LIN {X 0,Y 467.59,Z 413.241,A -85,B 0,C 180,E1 -7782.567,E2 -7782.567} C_VEL
LIN {X 0,Y 467.575,Z 413.244,A -85,B 0,C 180,E1 -7785.053,E2 -7785.053} C_VEL
LIN {X 0,Y 467.628,Z 413.238,A -85,B 0,C 180,E1 -7787.444,E2 -7787.444} C_VEL
LIN {X 0,Y 467.623,Z 413.239,A -85,B 0,C 180,E1 -7790.859,E2 -7790.859} C_VEL
LIN {X 0,Y 467.563,Z 413.244,A -85,B 0,C 180,E1 -7794.261,E2 -7794.261} C_VEL
LIN {X 0,Y 467.585,Z 413.242,A -85,B 0,C 180,E1 -7797.321,E2 -7797.321} C_VEL
LIN {X 0,Y 467.574,Z 413.245,A -85,B 0,C 180,E1 -7800.667,E2 -7800.667} C_VEL
LIN {X 0,Y 467.62,Z 413.238,A -85,B 0,C 180,E1 -7803.2,E2 -7803.2} C_VEL
LIN {X 0,Y 467.597,Z 413.241,A -85,B 0,C 180,E1 -7806.468,E2 -7806.468} C_VEL
LIN {X 0,Y 467.626,Z 413.235,A -85,B 0,C 180,E1 -7809.777,E2 -7809.777} C_VEL
LIN {X 0,Y 467.611,Z 413.24,A -85,B 0,C 180,E1 -7812.507,E2 -7812.507} C_VEL
LIN {X 0,Y 467.653,Z 413.233,A -85,B 0,C 180,E1 -7814.113,E2 -7814.113} C_VEL
LIN {X 0,Y 467.499,Z 414.001,A -85,B 0,C 180,E1 -7814.561,E2 -7814.561} C_VEL
LIN {X 0,Y 467.049,Z 415.884,A -85,B 0,C 180,E1 -7814.962,E2 -7814.962} C_VEL
LIN {X 0,Y 466.067,Z 420.004,A -85,B 0,C 180,E1 -7815.467,E2 -7815.467} C_VEL
LIN {X 0,Y 464.179,Z 429.024,A -85,B 0,C 180,E1 -7816.136,E2 -7816.136} C_VEL
LIN {X 0,Y 463.27,Z 436.592,A -85,B 0,C 180,E1 -7816.659,E2 -7816.659} C_VEL
LIN {X 0,Y 462.762,Z 447.595,A -85,B 0,C 180,E1 -7817.613,E2 -7817.613} C_VEL
LIN {X 0,Y 462.355,Z 456.798,A -85,B 0,C 180,E1 -7818.603,E2 -7818.603} C_VEL
LIN {X 0,Y 461.906,Z 465.182,A -85,B 0,C 180,E1 -7819.701,E2 -7819.701} C_VEL
LIN {X 0,Y 461.403,Z 473.311,A -85,B 0,C 180,E1 -7821.018,E2 -7821.018} C_VEL
LIN {X 0,Y 461.038,Z 479.446,A -85,B 0,C 180,E1 -7822.245,E2 -7822.245} C_VEL
LIN {X 0,Y 460.814,Z 485.803,A -85,B 0,C 180,E1 -7823.871,E2 -7823.871} C_VEL
LIN {X 0,Y 460.529,Z 489.69,A -85,B 0,C 180,E1 -7825.185,E2 -7825.185} C_VEL
LIN {X 0,Y 460.337,Z 492.556,A -85,B 0,C 180,E1 -7826.499,E2 -7826.499} C_VEL
LIN {X 0,Y 460.22,Z 493.935,A -85,B 0,C 180,E1 -7827.374,E2 -7827.374} C_VEL
LIN {X 0,Y 460.244,Z 494.899,A -85,B 0,C 180,E1 -7828.25,E2 -7828.25} C_VEL
LIN {X 0,Y 460.165,Z 495.736,A -85,B 0,C 180,E1 -7830,E2 -7830} C_VEL
LIN {X 0,Y 460.244,Z 494.978,A -85,B 0,C 180,E1 -7831.75,E2 -7831.75} C_VEL
LIN {X 0,Y 460.331,Z 492.716,A -85,B 0,C 180,E1 -7833.501,E2 -7833.501} C_VEL
LIN {X 0,Y 460.52,Z 489.91,A -85,B 0,C 180,E1 -7834.815,E2 -7834.815} C_VEL
LIN {X 0,Y 460.8,Z 486.099,A -85,B 0,C 180,E1 -7836.129,E2 -7836.129} C_VEL
LIN {X 0,Y 460.953,Z 480.215,A -85,B 0,C 180,E1 -7837.677,E2 -7837.677} C_VEL
LIN {X 0,Y 461.396,Z 473.809,A -85,B 0,C 180,E1 -7838.982,E2 -7838.982} C_VEL
LIN {X 0,Y 461.878,Z 465.789,A -85,B 0,C 180,E1 -7840.299,E2 -7840.299} C_VEL
LIN {X 0,Y 462.279,Z 457.573,A -85,B 0,C 180,E1 -7841.399,E2 -7841.399} C_VEL
LIN {X 0,Y 462.778,Z 447.396,A -85,B 0,C 180,E1 -7842.498,E2 -7842.498} C_VEL
LIN {X 0,Y 463.259,Z 436.893,A -85,B 0,C 180,E1 -7843.409,E2 -7843.409} C_VEL
LIN {X 0,Y 463.618,Z 426.234,A -85,B 0,C 180,E1 -7844.149,E2 -7844.149} C_VEL
LIN {X 0,Y 463.023,Z 422.562,A -85,B 0,C 180,E1 -7844.392,E2 -7844.392} C_VEL
LIN {X 0,Y 460.579,Z 414.111,A -85,B 0,C 180,E1 -7844.95,E2 -7844.95} C_VEL
LIN {X 0,Y 460.553,Z 414.12,A -85,B 0,C 180,E1 -7847.77,E2 -7847.77} C_VEL
LIN {X 0,Y 460.554,Z 414.117,A -85,B 0,C 180,E1 -7850.547,E2 -7850.547} C_VEL
LIN {X 0,Y 460.541,Z 414.12,A -85,B 0,C 180,E1 -7853.706,E2 -7853.706} C_VEL
LIN {X 0,Y 460.572,Z 414.114,A -85,B 0,C 180,E1 -7856.265,E2 -7856.265} C_VEL
LIN {X 0,Y 460.544,Z 414.12,A -85,B 0,C 180,E1 -7859.231,E2 -7859.231} C_VEL
LIN {X 0,Y 460.534,Z 414.118,A -85,B 0,C 180,E1 -7862.284,E2 -7862.284} C_VEL
LIN {X 0,Y 460.517,Z 414.123,A -85,B 0,C 180,E1 -7865.445,E2 -7865.445} C_VEL
LIN {X 0,Y 460.572,Z 414.116,A -85,B 0,C 180,E1 -7868.901,E2 -7868.901} C_VEL
LIN {X 0,Y 460.551,Z 414.116,A -85,B 0,C 180,E1 -7872.178,E2 -7872.178} C_VEL
LIN {X 0,Y 460.523,Z 414.122,A -85,B 0,C 180,E1 -7875.412,E2 -7875.412} C_VEL
LIN {X 0,Y 460.538,Z 414.119,A -85,B 0,C 180,E1 -7878.397,E2 -7878.397} C_VEL
LIN {X 0,Y 460.529,Z 414.121,A -85,B 0,C 180,E1 -7881.267,E2 -7881.267} C_VEL
LIN {X 0,Y 460.513,Z 414.123,A -85,B 0,C 180,E1 -7884.554,E2 -7884.554} C_VEL
LIN {X 0,Y 460.534,Z 414.118,A -85,B 0,C 180,E1 -7887.716,E2 -7887.716} C_VEL
LIN {X 0,Y 460.543,Z 414.12,A -85,B 0,C 180,E1 -7890.769,E2 -7890.769} C_VEL
LIN {X 0,Y 460.559,Z 414.115,A -85,B 0,C 180,E1 -7893.734,E2 -7893.734} C_VEL
LIN {X 0,Y 460.547,Z 414.12,A -85,B 0,C 180,E1 -7896.624,E2 -7896.624} C_VEL
LIN {X 0,Y 460.555,Z 414.116,A -85,B 0,C 180,E1 -7899.453,E2 -7899.453} C_VEL
LIN {X 0,Y 460.563,Z 414.118,A -85,B 0,C 180,E1 -7902.23,E2 -7902.23} C_VEL
LIN {X 0,Y 460.569,Z 414.117,A -85,B 0,C 180,E1 -7904.965,E2 -7904.965} C_VEL
LIN {X 0,Y 460.633,Z 414.106,A -85,B 0,C 180,E1 -7907.666,E2 -7907.666} C_VEL
LIN {X 0,Y 460.623,Z 414.108,A -85,B 0,C 180,E1 -7911.224,E2 -7911.224} C_VEL
LIN {X 0,Y 460.71,Z 414.098,A -85,B 0,C 180,E1 -7913.87,E2 -7913.87} C_VEL
LIN {X 0,Y 460.828,Z 414.081,A -85,B 0,C 180,E1 -7917.378,E2 -7917.378} C_VEL
LIN {X 0,Y 460.857,Z 414.08,A -85,B 0,C 180,E1 -7920,E2 -7920} C_VEL
LIN {X 0,Y 460.829,Z 414.084,A -85,B 0,C 180,E1 -7922.622,E2 -7922.622} C_VEL
LIN {X 0,Y 460.711,Z 414.099,A -85,B 0,C 180,E1 -7926.13,E2 -7926.13} C_VEL
LIN {X 0,Y 460.622,Z 414.109,A -85,B 0,C 180,E1 -7928.776,E2 -7928.776} C_VEL
LIN {X 0,Y 460.637,Z 414.109,A -85,B 0,C 180,E1 -7932.457,E2 -7932.457} C_VEL
LIN {X 0,Y 460.603,Z 414.114,A -85,B 0,C 180,E1 -7935.997,E2 -7935.997} C_VEL
LIN {X 0,Y 460.574,Z 414.114,A -85,B 0,C 180,E1 -7938.902,E2 -7938.902} C_VEL
LIN {X 0,Y 460.518,Z 414.122,A -85,B 0,C 180,E1 -7941.486,E2 -7941.486} C_VEL
LIN {X 0,Y 460.533,Z 414.121,A -85,B 0,C 180,E1 -7944.333,E2 -7944.333} C_VEL
LIN {X 0,Y 460.591,Z 414.115,A -85,B 0,C 180,E1 -7947.748,E2 -7947.748} C_VEL
LIN {X 0,Y 460.525,Z 414.12,A -85,B 0,C 180,E1 -7951.283,E2 -7951.283} C_VEL
LIN {X 0,Y 460.536,Z 414.12,A -85,B 0,C 180,E1 -7954.506,E2 -7954.506} C_VEL
LIN {X 0,Y 460.53,Z 414.121,A -85,B 0,C 180,E1 -7957.62,E2 -7957.62} C_VEL
LIN {X 0,Y 460.545,Z 414.119,A -85,B 0,C 180,E1 -7960.27,E2 -7960.27} C_VEL
LIN {X 0,Y 460.511,Z 414.125,A -85,B 0,C 180,E1 -7963.374,E2 -7963.374} C_VEL
LIN {X 0,Y 460.502,Z 414.127,A -85,B 0,C 180,E1 -7966.625,E2 -7966.625} C_VEL
LIN {X 0,Y 460.577,Z 414.173,A -85,B 0,C 180,E1 -7969.496,E2 -7969.496} C_VEL
LIN {X 0,Y 462.384,Z 423.509,A -85,B 0,C 180,E1 -7972.221,E2 -7972.221} C_VEL
LIN {X 0,Y 463.139,Z 428.94,A -85,B 0,C 180,E1 -7973.714,E2 -7973.714} C_VEL
LIN {X 0,Y 462.392,Z 443.333,A -85,B 0,C 180,E1 -7977.345,E2 -7977.345} C_VEL
LIN {X 0,Y 461.898,Z 456.337,A -85,B 0,C 180,E1 -7980.501,E2 -7980.501} C_VEL
LIN {X 0,Y 461.394,Z 471.111,A -85,B 0,C 180,E1 -7983.987,E2 -7983.987} C_VEL
LIN {X 0,Y 460.935,Z 485.612,A -85,B 0,C 180,E1 -7987.357,E2 -7987.357} C_VEL
LIN {X 0,Y 460.576,Z 500.515,A -85,B 0,C 180,E1 -7990.799,E2 -7990.799} C_VEL
LIN {X 0,Y 460.234,Z 515.613,A -85,B 0,C 180,E1 -7994.309,E2 -7994.309} C_VEL
LIN {X 0,Y 461.616,Z 530.277,A -85,B 0,C 180,E1 -7994.719,E2 -7994.719} C_VEL
LIN {X 0,Y 462.685,Z 543.371,A -85,B 0,C 180,E1 -7995.26,E2 -7995.26} C_VEL
LIN {X 0,Y 462.165,Z 555.697,A -85,B 0,C 180,E1 -7995.918,E2 -7995.918} C_VEL
LIN {X 0,Y 461.571,Z 568.295,A -85,B 0,C 180,E1 -7996.797,E2 -7996.797} C_VEL
LIN {X 0,Y 461.172,Z 579.391,A -85,B 0,C 180,E1 -7997.793,E2 -7997.793} C_VEL
LIN {X 0,Y 460.671,Z 588.435,A -85,B 0,C 180,E1 -7998.784,E2 -7998.784} C_VEL
LIN {X 0,Y 460.277,Z 598.303,A -85,B 0,C 180,E1 -8000.109,E2 -8000.109} C_VEL
LIN {X 0,Y 460.041,Z 606.193,A -85,B 0,C 180,E1 -8001.434,E2 -8001.434} C_VEL
LIN {X 0,Y 459.919,Z 613.486,A -85,B 0,C 180,E1 -8002.978,E2 -8002.978} C_VEL
LIN {X 0,Y 459.902,Z 618.355,A -85,B 0,C 180,E1 -8004.299,E2 -8004.299} C_VEL
LIN {X 0,Y 459.908,Z 622.081,A -85,B 0,C 180,E1 -8005.618,E2 -8005.618} C_VEL
LIN {X 0,Y 459.916,Z 624.005,A -85,B 0,C 180,E1 -8006.496,E2 -8006.496} C_VEL
LIN {X 0,Y 459.908,Z 625.446,A -85,B 0,C 180,E1 -8007.372,E2 -8007.372} C_VEL
LIN {X 0,Y 459.889,Z 626.473,A -85,B 0,C 180,E1 -8008.249,E2 -8008.249} C_VEL
LIN {X 0,Y 460.003,Z 627.34,A -85,B 0,C 180,E1 -8010,E2 -8010} C_VEL
LIN {X 0,Y 459.889,Z 626.474,A -85,B 0,C 180,E1 -8011.752,E2 -8011.752} C_VEL
LIN {X 0,Y 459.908,Z 625.45,A -85,B 0,C 180,E1 -8012.628,E2 -8012.628} C_VEL
LIN {X 0,Y 459.916,Z 624.008,A -85,B 0,C 180,E1 -8013.504,E2 -8013.504} C_VEL
LIN {X 0,Y 459.907,Z 620.977,A -85,B 0,C 180,E1 -8014.821,E2 -8014.821} C_VEL
LIN {X 0,Y 459.934,Z 616.882,A -85,B 0,C 180,E1 -8016.14,E2 -8016.14} C_VEL
LIN {X 0,Y 459.968,Z 610.586,A -85,B 0,C 180,E1 -8017.683,E2 -8017.683} C_VEL
LIN {X 0,Y 460.103,Z 603.731,A -85,B 0,C 180,E1 -8019.008,E2 -8019.008} C_VEL
LIN {X 0,Y 460.368,Z 595.255,A -85,B 0,C 180,E1 -8020.334,E2 -8020.334} C_VEL
LIN {X 0,Y 460.718,Z 586.591,A -85,B 0,C 180,E1 -8021.438,E2 -8021.438} C_VEL
LIN {X 0,Y 461.257,Z 576.549,A -85,B 0,C 180,E1 -8022.483,E2 -8022.483} C_VEL
LIN {X 0,Y 461.652,Z 566.849,A -85,B 0,C 180,E1 -8023.312,E2 -8023.312} C_VEL
LIN {X 0,Y 462.156,Z 555.684,A -85,B 0,C 180,E1 -8024.082,E2 -8024.082} C_VEL
LIN {X 0,Y 462.704,Z 543.348,A -85,B 0,C 180,E1 -8024.739,E2 -8024.739} C_VEL
LIN {X 0,Y 461.648,Z 530.24,A -85,B 0,C 180,E1 -8025.28,E2 -8025.28} C_VEL
LIN {X 0,Y 460.202,Z 515.503,A -85,B 0,C 180,E1 -8025.714,E2 -8025.714} C_VEL
LIN {X 0,Y 460.55,Z 501.845,A -85,B 0,C 180,E1 -8028.893,E2 -8028.893} C_VEL
LIN {X 0,Y 460.919,Z 486.637,A -85,B 0,C 180,E1 -8032.408,E2 -8032.408} C_VEL
LIN {X 0,Y 461.353,Z 472.748,A -85,B 0,C 180,E1 -8035.628,E2 -8035.628} C_VEL
LIN {X 0,Y 461.814,Z 457.82,A -85,B 0,C 180,E1 -8039.143,E2 -8039.143} C_VEL
LIN {X 0,Y 462.292,Z 445.378,A -85,B 0,C 180,E1 -8042.147,E2 -8042.147} C_VEL
LIN {X 0,Y 463.049,Z 430.956,A -85,B 0,C 180,E1 -8045.757,E2 -8045.757} C_VEL
LIN {X 0,Y 462.961,Z 426.694,A -85,B 0,C 180,E1 -8046.88,E2 -8046.88} C_VEL
LIN {X 0,Y 461.063,Z 416.459,A -85,B 0,C 180,E1 -8049.808,E2 -8049.808} C_VEL
LIN {X 0,Y 460.577,Z 414.114,A -85,B 0,C 180,E1 -8050.554,E2 -8050.554} C_VEL
LIN {X 0,Y 460.503,Z 414.123,A -85,B 0,C 180,E1 -8053.375,E2 -8053.375} C_VEL
LIN {X 0,Y 460.512,Z 414.126,A -85,B 0,C 180,E1 -8056.626,E2 -8056.626} C_VEL
LIN {X 0,Y 460.546,Z 414.119,A -85,B 0,C 180,E1 -8059.73,E2 -8059.73} C_VEL
LIN {X 0,Y 460.53,Z 414.121,A -85,B 0,C 180,E1 -8062.519,E2 -8062.519} C_VEL
LIN {X 0,Y 460.552,Z 414.118,A -85,B 0,C 180,E1 -8065.624,E2 -8065.624} C_VEL
LIN {X 0,Y 460.54,Z 414.118,A -85,B 0,C 180,E1 -8068.745,E2 -8068.745} C_VEL
LIN {X 0,Y 460.592,Z 414.115,A -85,B 0,C 180,E1 -8072.252,E2 -8072.252} C_VEL
LIN {X 0,Y 460.534,Z 414.121,A -85,B 0,C 180,E1 -8075.667,E2 -8075.667} C_VEL
LIN {X 0,Y 460.525,Z 414.121,A -85,B 0,C 180,E1 -8078.578,E2 -8078.578} C_VEL
LIN {X 0,Y 460.595,Z 414.113,A -85,B 0,C 180,E1 -8081.311,E2 -8081.311} C_VEL
LIN {X 0,Y 460.608,Z 414.113,A -85,B 0,C 180,E1 -8084.059,E2 -8084.059} C_VEL
LIN {X 0,Y 460.634,Z 414.109,A -85,B 0,C 180,E1 -8087.667,E2 -8087.667} C_VEL
LIN {X 0,Y 460.623,Z 414.109,A -85,B 0,C 180,E1 -8091.224,E2 -8091.224} C_VEL
LIN {X 0,Y 460.712,Z 414.099,A -85,B 0,C 180,E1 -8093.87,E2 -8093.87} C_VEL
LIN {X 0,Y 460.83,Z 414.084,A -85,B 0,C 180,E1 -8097.378,E2 -8097.378} C_VEL
LIN {X 0,Y 460.858,Z 414.08,A -85,B 0,C 180,E1 -8100,E2 -8100} C_VEL
LIN {X 0,Y 460.805,Z 414.084,A -85,B 0,C 180,E1 -8102.623,E2 -8102.623} C_VEL
LIN {X 0,Y 460.706,Z 414.099,A -85,B 0,C 180,E1 -8106.13,E2 -8106.13} C_VEL
LIN {X 0,Y 460.625,Z 414.108,A -85,B 0,C 180,E1 -8108.776,E2 -8108.776} C_VEL
LIN {X 0,Y 460.638,Z 414.105,A -85,B 0,C 180,E1 -8112.457,E2 -8112.457} C_VEL
LIN {X 0,Y 460.604,Z 414.111,A -85,B 0,C 180,E1 -8115.998,E2 -8115.998} C_VEL
LIN {X 0,Y 460.575,Z 414.115,A -85,B 0,C 180,E1 -8118.902,E2 -8118.902} C_VEL
LIN {X 0,Y 460.52,Z 414.123,A -85,B 0,C 180,E1 -8121.486,E2 -8121.486} C_VEL
LIN {X 0,Y 460.545,Z 414.117,A -85,B 0,C 180,E1 -8124.332,E2 -8124.332} C_VEL
LIN {X 0,Y 460.583,Z 414.115,A -85,B 0,C 180,E1 -8127.243,E2 -8127.243} C_VEL
LIN {X 0,Y 460.515,Z 414.12,A -85,B 0,C 180,E1 -8130.24,E2 -8130.24} C_VEL
LIN {X 0,Y 460.533,Z 414.121,A -85,B 0,C 180,E1 -8133.325,E2 -8133.325} C_VEL
LIN {X 0,Y 460.48,Z 414.127,A -85,B 0,C 180,E1 -8136.529,E2 -8136.529} C_VEL
LIN {X 0,Y 460.531,Z 414.119,A -85,B 0,C 180,E1 -8139.863,E2 -8139.863} C_VEL
LIN {X 0,Y 460.521,Z 414.123,A -85,B 0,C 180,E1 -8142.901,E2 -8142.901} C_VEL
LIN {X 0,Y 460.528,Z 414.119,A -85,B 0,C 180,E1 -8145.829,E2 -8145.829} C_VEL
LIN {X 0,Y 460.547,Z 414.12,A -85,B 0,C 180,E1 -8148.99,E2 -8148.99} C_VEL
LIN {X 0,Y 460.551,Z 414.119,A -85,B 0,C 180,E1 -8151.269,E2 -8151.269} C_VEL
LIN {X 0,Y 460.514,Z 414.124,A -85,B 0,C 180,E1 -8154.554,E2 -8154.554} C_VEL
LIN {X 0,Y 460.535,Z 414.118,A -85,B 0,C 180,E1 -8157.716,E2 -8157.716} C_VEL
LIN {X 0,Y 460.544,Z 414.121,A -85,B 0,C 180,E1 -8160.769,E2 -8160.769} C_VEL
LIN {X 0,Y 460.567,Z 414.115,A -85,B 0,C 180,E1 -8163.735,E2 -8163.735} C_VEL
LIN {X 0,Y 460.55,Z 414.119,A -85,B 0,C 180,E1 -8166.624,E2 -8166.624} C_VEL
LIN {X 0,Y 460.555,Z 414.117,A -85,B 0,C 180,E1 -8169.453,E2 -8169.453} C_VEL
LIN {X 0,Y 460.562,Z 414.119,A -85,B 0,C 180,E1 -8172.23,E2 -8172.23} C_VEL
LIN {X 0,Y 460.588,Z 414.114,A -85,B 0,C 180,E1 -8175.163,E2 -8175.163} C_VEL
LIN {X 0,Y 463.568,Z 424.775,A -85,B 0,C 180,E1 -8175.85,E2 -8175.85} C_VEL
LIN {X 0,Y 463.27,Z 436.592,A -85,B 0,C 180,E1 -8176.659,E2 -8176.659} C_VEL
LIN {X 0,Y 462.41,Z 441.639,A -85,B 0,C 180,E1 -8177.041,E2 -8177.041} C_VEL
LIN {X 0,Y 459.31,Z 449.618,A -85,B 0,C 180,E1 -8177.669,E2 -8177.669} C_VEL
LIN {X 0,Y 456.17,Z 457.098,A -85,B 0,C 180,E1 -8178.374,E2 -8178.374} C_VEL
LIN {X 0,Y 455.248,Z 461.313,A -85,B 0,C 180,E1 -8178.869,E2 -8178.869} C_VEL
LIN {X 0,Y 454.813,Z 469.099,A -85,B 0,C 180,E1 -8179.989,E2 -8179.989} C_VEL
LIN {X 0,Y 454.314,Z 476.678,A -85,B 0,C 180,E1 -8181.325,E2 -8181.325} C_VEL
LIN {X 0,Y 454.066,Z 481.966,A -85,B 0,C 180,E1 -8182.475,E2 -8182.475} C_VEL
LIN {X 0,Y 453.838,Z 486.808,A -85,B 0,C 180,E1 -8183.777,E2 -8183.777} C_VEL
LIN {X 0,Y 453.526,Z 490.696,A -85,B 0,C 180,E1 -8185.111,E2 -8185.111} C_VEL
LIN {X 0,Y 453.322,Z 493.562,A -85,B 0,C 180,E1 -8186.445,E2 -8186.445} C_VEL
LIN {X 0,Y 453.2,Z 494.941,A -85,B 0,C 180,E1 -8187.333,E2 -8187.333} C_VEL
LIN {X 0,Y 453.225,Z 495.903,A -85,B 0,C 180,E1 -8188.223,E2 -8188.223} C_VEL
LIN {X 0,Y 453.163,Z 496.737,A -85,B 0,C 180,E1 -8190,E2 -8190} C_VEL
LIN {X 0,Y 453.224,Z 495.982,A -85,B 0,C 180,E1 -8191.777,E2 -8191.777} C_VEL
LIN {X 0,Y 453.315,Z 493.721,A -85,B 0,C 180,E1 -8193.555,E2 -8193.555} C_VEL
LIN {X 0,Y 453.518,Z 490.914,A -85,B 0,C 180,E1 -8194.889,E2 -8194.889} C_VEL
LIN {X 0,Y 453.824,Z 487.101,A -85,B 0,C 180,E1 -8196.223,E2 -8196.223} C_VEL
LIN {X 0,Y 453.989,Z 481.22,A -85,B 0,C 180,E1 -8197.795,E2 -8197.795} C_VEL
LIN {X 0,Y 454.457,Z 474.811,A -85,B 0,C 180,E1 -8199.121,E2 -8199.121} C_VEL
LIN {X 0,Y 454.967,Z 466.791,A -85,B 0,C 180,E1 -8200.457,E2 -8200.457} C_VEL
LIN {X 0,Y 455.394,Z 458.574,A -85,B 0,C 180,E1 -8201.574,E2 -8201.574} C_VEL
LIN {X 0,Y 455.919,Z 448.396,A -85,B 0,C 180,E1 -8202.689,E2 -8202.689} C_VEL
LIN {X 0,Y 456.426,Z 437.892,A -85,B 0,C 180,E1 -8203.613,E2 -8203.613} C_VEL
LIN {X 0,Y 456.794,Z 427.234,A -85,B 0,C 180,E1 -8204.365,E2 -8204.365} C_VEL
LIN {X 0,Y 455.182,Z 420.664,A -85,B 0,C 180,E1 -8204.82,E2 -8204.82} C_VEL
LIN {X 0,Y 453.537,Z 414.991,A -85,B 0,C 180,E1 -8205.188,E2 -8205.188} C_VEL
LIN {X 0,Y 453.507,Z 414.997,A -85,B 0,C 180,E1 -8208.056,E2 -8208.056} C_VEL
LIN {X 0,Y 453.486,Z 414.998,A -85,B 0,C 180,E1 -8210.882,E2 -8210.882} C_VEL
LIN {X 0,Y 453.503,Z 414.996,A -85,B 0,C 180,E1 -8213.889,E2 -8213.889} C_VEL
LIN {X 0,Y 453.517,Z 414.994,A -85,B 0,C 180,E1 -8216.705,E2 -8216.705} C_VEL
LIN {X 0,Y 453.476,Z 414.998,A -85,B 0,C 180,E1 -8219.785,E2 -8219.785} C_VEL
LIN {X 0,Y 453.493,Z 414.998,A -85,B 0,C 180,E1 -8223.189,E2 -8223.189} C_VEL
LIN {X 0,Y 453.459,Z 415,A -85,B 0,C 180,E1 -8226.3,E2 -8226.3} C_VEL
LIN {X 0,Y 453.536,Z 414.992,A -85,B 0,C 180,E1 -8229.445,E2 -8229.445} C_VEL
LIN {X 0,Y 453.495,Z 414.998,A -85,B 0,C 180,E1 -8232.991,E2 -8232.991} C_VEL
LIN {X 0,Y 453.476,Z 414.997,A -85,B 0,C 180,E1 -8235.78,E2 -8235.78} C_VEL
LIN {X 0,Y 453.484,Z 414.997,A -85,B 0,C 180,E1 -8238.21,E2 -8238.21} C_VEL
LIN {X 0,Y 453.512,Z 414.997,A -85,B 0,C 180,E1 -8240.791,E2 -8240.791} C_VEL
LIN {X 0,Y 453.457,Z 415,A -85,B 0,C 180,E1 -8243.917,E2 -8243.917} C_VEL
LIN {X 0,Y 453.485,Z 414.999,A -85,B 0,C 180,E1 -8247.151,E2 -8247.151} C_VEL
LIN {X 0,Y 453.478,Z 414.998,A -85,B 0,C 180,E1 -8250.268,E2 -8250.268} C_VEL
LIN {X 0,Y 453.508,Z 414.995,A -85,B 0,C 180,E1 -8253.294,E2 -8253.294} C_VEL
LIN {X 0,Y 453.5,Z 414.996,A -85,B 0,C 180,E1 -8256.238,E2 -8256.238} C_VEL
LIN {X 0,Y 453.486,Z 414.998,A -85,B 0,C 180,E1 -8259.118,E2 -8259.118} C_VEL
LIN {X 0,Y 453.515,Z 414.993,A -85,B 0,C 180,E1 -8261.945,E2 -8261.945} C_VEL
LIN {X 0,Y 453.543,Z 414.992,A -85,B 0,C 180,E1 -8264.726,E2 -8264.726} C_VEL
LIN {X 0,Y 453.605,Z 414.981,A -85,B 0,C 180,E1 -8267.472,E2 -8267.472} C_VEL
LIN {X 0,Y 453.589,Z 414.985,A -85,B 0,C 180,E1 -8271.086,E2 -8271.086} C_VEL
LIN {X 0,Y 453.676,Z 414.973,A -85,B 0,C 180,E1 -8273.775,E2 -8273.775} C_VEL
LIN {X 0,Y 453.768,Z 414.961,A -85,B 0,C 180,E1 -8277.337,E2 -8277.337} C_VEL
LIN {X 0,Y 453.827,Z 414.956,A -85,B 0,C 180,E1 -8280,E2 -8280} C_VEL
LIN {X 0,Y 453.769,Z 414.964,A -85,B 0,C 180,E1 -8282.663,E2 -8282.663} C_VEL
LIN {X 0,Y 453.677,Z 414.976,A -85,B 0,C 180,E1 -8286.225,E2 -8286.225} C_VEL
LIN {X 0,Y 453.588,Z 414.985,A -85,B 0,C 180,E1 -8288.913,E2 -8288.913} C_VEL
LIN {X 0,Y 453.605,Z 414.984,A -85,B 0,C 180,E1 -8292.551,E2 -8292.551} C_VEL
LIN {X 0,Y 453.547,Z 414.992,A -85,B 0,C 180,E1 -8296.196,E2 -8296.196} C_VEL
LIN {X 0,Y 453.524,Z 414.992,A -85,B 0,C 180,E1 -8299.041,E2 -8299.041} C_VEL
LIN {X 0,Y 453.479,Z 415,A -85,B 0,C 180,E1 -8301.836,E2 -8301.836} C_VEL
LIN {X 0,Y 453.503,Z 414.995,A -85,B 0,C 180,E1 -8304.735,E2 -8304.735} C_VEL
LIN {X 0,Y 453.54,Z 414.993,A -85,B 0,C 180,E1 -8307.961,E2 -8307.961} C_VEL
LIN {X 0,Y 453.469,Z 415,A -85,B 0,C 180,E1 -8311.525,E2 -8311.525} C_VEL
LIN {X 0,Y 453.491,Z 414.996,A -85,B 0,C 180,E1 -8314.778,E2 -8314.778} C_VEL
LIN {X 0,Y 453.475,Z 414.999,A -85,B 0,C 180,E1 -8318.311,E2 -8318.311} C_VEL
LIN {X 0,Y 453.496,Z 414.995,A -85,B 0,C 180,E1 -8320.609,E2 -8320.609} C_VEL
LIN {X 0,Y 453.466,Z 415.003,A -85,B 0,C 180,E1 -8323.245,E2 -8323.245} C_VEL
LIN {X 0,Y 453.468,Z 415,A -85,B 0,C 180,E1 -8325.779,E2 -8325.779} C_VEL
LIN {X 0,Y 453.547,Z 415.09,A -85,B 0,C 180,E1 -8329.215,E2 -8329.215} C_VEL
LIN {X 0,Y 455.304,Z 424.201,A -85,B 0,C 180,E1 -8331.927,E2 -8331.927} C_VEL
LIN {X 0,Y 456.117,Z 428.865,A -85,B 0,C 180,E1 -8333.248,E2 -8333.248} C_VEL
LIN {X 0,Y 455.896,Z 434.726,A -85,B 0,C 180,E1 -8334.79,E2 -8334.79} C_VEL
LIN {X 0,Y 455.244,Z 448.739,A -85,B 0,C 180,E1 -8338.339,E2 -8338.339} C_VEL
LIN {X 0,Y 454.736,Z 461.139,A -85,B 0,C 180,E1 -8341.373,E2 -8341.373} C_VEL
LIN {X 0,Y 454.24,Z 474.519,A -85,B 0,C 180,E1 -8344.574,E2 -8344.574} C_VEL
LIN {X 0,Y 453.833,Z 487.75,A -85,B 0,C 180,E1 -8347.703,E2 -8347.703} C_VEL
LIN {X 0,Y 453.486,Z 501.768,A -85,B 0,C 180,E1 -8351.007,E2 -8351.007} C_VEL
LIN {X 0,Y 453.143,Z 514.766,A -85,B 0,C 180,E1 -8354.068,E2 -8354.068} C_VEL
LIN {X 0,Y 454.552,Z 528.842,A -85,B 0,C 180,E1 -8354.463,E2 -8354.463} C_VEL
LIN {X 0,Y 455.427,Z 539.753,A -85,B 0,C 180,E1 -8354.906,E2 -8354.906} C_VEL
LIN {X 0,Y 455.703,Z 544.635,A -85,B 0,C 180,E1 -8355.144,E2 -8355.144} C_VEL
LIN {X 0,Y 455.135,Z 556.46,A -85,B 0,C 180,E1 -8355.81,E2 -8355.81} C_VEL
LIN {X 0,Y 454.606,Z 567.274,A -85,B 0,C 180,E1 -8356.591,E2 -8356.591} C_VEL
LIN {X 0,Y 454.174,Z 578.369,A -85,B 0,C 180,E1 -8357.602,E2 -8357.602} C_VEL
LIN {X 0,Y 453.643,Z 587.412,A -85,B 0,C 180,E1 -8358.608,E2 -8358.608} C_VEL
LIN {X 0,Y 453.212,Z 597.279,A -85,B 0,C 180,E1 -8359.953,E2 -8359.953} C_VEL
LIN {X 0,Y 452.974,Z 605.172,A -85,B 0,C 180,E1 -8361.299,E2 -8361.299} C_VEL
LIN {X 0,Y 452.87,Z 610.593,A -85,B 0,C 180,E1 -8362.42,E2 -8362.42} C_VEL
LIN {X 0,Y 452.85,Z 615.865,A -85,B 0,C 180,E1 -8363.763,E2 -8363.763} C_VEL
LIN {X 0,Y 452.859,Z 619.965,A -85,B 0,C 180,E1 -8365.104,E2 -8365.104} C_VEL
LIN {X 0,Y 452.873,Z 622.996,A -85,B 0,C 180,E1 -8366.441,E2 -8366.441} C_VEL
LIN {X 0,Y 452.866,Z 624.438,A -85,B 0,C 180,E1 -8367.332,E2 -8367.332} C_VEL
LIN {X 0,Y 452.854,Z 625.466,A -85,B 0,C 180,E1 -8368.221,E2 -8368.221} C_VEL
LIN {X 0,Y 452.986,Z 626.337,A -85,B 0,C 180,E1 -8370,E2 -8370} C_VEL
LIN {X 0,Y 452.854,Z 625.468,A -85,B 0,C 180,E1 -8371.779,E2 -8371.779} C_VEL
LIN {X 0,Y 452.866,Z 624.441,A -85,B 0,C 180,E1 -8372.669,E2 -8372.669} C_VEL
LIN {X 0,Y 452.873,Z 622.999,A -85,B 0,C 180,E1 -8373.559,E2 -8373.559} C_VEL
LIN {X 0,Y 452.859,Z 619.966,A -85,B 0,C 180,E1 -8374.897,E2 -8374.897} C_VEL
LIN {X 0,Y 452.847,Z 615.862,A -85,B 0,C 180,E1 -8376.237,E2 -8376.237} C_VEL
LIN {X 0,Y 452.901,Z 609.565,A -85,B 0,C 180,E1 -8377.804,E2 -8377.804} C_VEL
LIN {X 0,Y 453.065,Z 602.711,A -85,B 0,C 180,E1 -8379.149,E2 -8379.149} C_VEL
LIN {X 0,Y 453.331,Z 594.231,A -85,B 0,C 180,E1 -8380.496,E2 -8380.496} C_VEL
LIN {X 0,Y 453.684,Z 585.563,A -85,B 0,C 180,E1 -8381.618,E2 -8381.618} C_VEL
LIN {X 0,Y 454.216,Z 576.067,A -85,B 0,C 180,E1 -8382.627,E2 -8382.627} C_VEL
LIN {X 0,Y 454.78,Z 564.38,A -85,B 0,C 180,E1 -8383.631,E2 -8383.631} C_VEL
LIN {X 0,Y 455.328,Z 552.874,A -85,B 0,C 180,E1 -8384.412,E2 -8384.412} C_VEL
LIN {X 0,Y 455.732,Z 542.312,A -85,B 0,C 180,E1 -8384.97,E2 -8384.97} C_VEL
LIN {X 0,Y 454.69,Z 530.257,A -85,B 0,C 180,E1 -8385.487,E2 -8385.487} C_VEL
LIN {X 0,Y 453.321,Z 516.581,A -85,B 0,C 180,E1 -8385.89,E2 -8385.89} C_VEL
LIN {X 0,Y 453.151,Z 514.574,A -85,B 0,C 180,E1 -8385.943,E2 -8385.943} C_VEL
LIN {X 0,Y 453.515,Z 499.972,A -85,B 0,C 180,E1 -8389.415,E2 -8389.415} C_VEL
LIN {X 0,Y 453.931,Z 484.708,A -85,B 0,C 180,E1 -8393.013,E2 -8393.013} C_VEL
LIN {X 0,Y 454.337,Z 471.213,A -85,B 0,C 180,E1 -8396.209,E2 -8396.209} C_VEL
LIN {X 0,Y 454.851,Z 458.02,A -85,B 0,C 180,E1 -8399.379,E2 -8399.379} C_VEL
LIN {X 0,Y 455.32,Z 446.381,A -85,B 0,C 180,E1 -8402.242,E2 -8402.242} C_VEL
LIN {X 0,Y 456.098,Z 432.25,A -85,B 0,C 180,E1 -8405.841,E2 -8405.841} C_VEL
LIN {X 0,Y 456.016,Z 428.134,A -85,B 0,C 180,E1 -8406.946,E2 -8406.946} C_VEL
LIN {X 0,Y 454.094,Z 417.758,A -85,B 0,C 180,E1 -8409.963,E2 -8409.963} C_VEL
LIN {X 0,Y 453.52,Z 414.995,A -85,B 0,C 180,E1 -8410.818,E2 -8410.818} C_VEL
LIN {X 0,Y 453.49,Z 415,A -85,B 0,C 180,E1 -8414.529,E2 -8414.529} C_VEL
LIN {X 0,Y 453.481,Z 415,A -85,B 0,C 180,E1 -8418.065,E2 -8418.065} C_VEL
LIN {X 0,Y 453.513,Z 414.994,A -85,B 0,C 180,E1 -8420.791,E2 -8420.791} C_VEL
LIN {X 0,Y 453.46,Z 415.003,A -85,B 0,C 180,E1 -8423.918,E2 -8423.918} C_VEL
LIN {X 0,Y 453.487,Z 414.996,A -85,B 0,C 180,E1 -8427.151,E2 -8427.151} C_VEL
LIN {X 0,Y 453.479,Z 415,A -85,B 0,C 180,E1 -8430.269,E2 -8430.269} C_VEL
LIN {X 0,Y 453.508,Z 414.994,A -85,B 0,C 180,E1 -8433.294,E2 -8433.294} C_VEL
LIN {X 0,Y 453.501,Z 414.997,A -85,B 0,C 180,E1 -8436.239,E2 -8436.239} C_VEL
LIN {X 0,Y 453.487,Z 414.997,A -85,B 0,C 180,E1 -8439.118,E2 -8439.118} C_VEL
LIN {X 0,Y 453.517,Z 414.997,A -85,B 0,C 180,E1 -8441.945,E2 -8441.945} C_VEL
LIN {X 0,Y 453.544,Z 414.988,A -85,B 0,C 180,E1 -8444.726,E2 -8444.726} C_VEL
LIN {X 0,Y 453.606,Z 414.984,A -85,B 0,C 180,E1 -8447.472,E2 -8447.472} C_VEL
LIN {X 0,Y 453.589,Z 414.984,A -85,B 0,C 180,E1 -8451.087,E2 -8451.087} C_VEL
LIN {X 0,Y 453.678,Z 414.976,A -85,B 0,C 180,E1 -8453.775,E2 -8453.775} C_VEL
LIN {X 0,Y 453.77,Z 414.964,A -85,B 0,C 180,E1 -8457.337,E2 -8457.337} C_VEL
LIN {X 0,Y 453.828,Z 414.956,A -85,B 0,C 180,E1 -8460,E2 -8460} C_VEL
LIN {X 0,Y 453.749,Z 414.963,A -85,B 0,C 180,E1 -8462.663,E2 -8462.663} C_VEL
LIN {X 0,Y 453.673,Z 414.974,A -85,B 0,C 180,E1 -8466.225,E2 -8466.225} C_VEL
LIN {X 0,Y 453.591,Z 414.985,A -85,B 0,C 180,E1 -8468.913,E2 -8468.913} C_VEL
LIN {X 0,Y 453.606,Z 414.981,A -85,B 0,C 180,E1 -8472.551,E2 -8472.551} C_VEL
LIN {X 0,Y 453.549,Z 414.988,A -85,B 0,C 180,E1 -8476.196,E2 -8476.196} C_VEL
LIN {X 0,Y 453.525,Z 414.994,A -85,B 0,C 180,E1 -8479.041,E2 -8479.041} C_VEL
LIN {X 0,Y 453.48,Z 414.999,A -85,B 0,C 180,E1 -8481.836,E2 -8481.836} C_VEL
LIN {X 0,Y 453.517,Z 414.994,A -85,B 0,C 180,E1 -8484.734,E2 -8484.734} C_VEL
LIN {X 0,Y 453.541,Z 414.99,A -85,B 0,C 180,E1 -8487.961,E2 -8487.961} C_VEL
LIN {X 0,Y 453.471,Z 415.001,A -85,B 0,C 180,E1 -8491.525,E2 -8491.525} C_VEL
LIN {X 0,Y 453.491,Z 414.997,A -85,B 0,C 180,E1 -8494.777,E2 -8494.777} C_VEL
LIN {X 0,Y 453.466,Z 414.999,A -85,B 0,C 180,E1 -8498.312,E2 -8498.312} C_VEL
LIN {X 0,Y 453.497,Z 414.997,A -85,B 0,C 180,E1 -8500.609,E2 -8500.609} C_VEL
LIN {X 0,Y 453.467,Z 415.002,A -85,B 0,C 180,E1 -8503.245,E2 -8503.245} C_VEL
LIN {X 0,Y 453.481,Z 414.997,A -85,B 0,C 180,E1 -8505.78,E2 -8505.78} C_VEL
LIN {X 0,Y 453.5,Z 414.995,A -85,B 0,C 180,E1 -8508.211,E2 -8508.211} C_VEL
LIN {X 0,Y 453.536,Z 414.993,A -85,B 0,C 180,E1 -8510.787,E2 -8510.787} C_VEL
LIN {X 0,Y 453.458,Z 415,A -85,B 0,C 180,E1 -8513.917,E2 -8513.917} C_VEL
LIN {X 0,Y 453.486,Z 415,A -85,B 0,C 180,E1 -8517.151,E2 -8517.151} C_VEL
LIN {X 0,Y 453.479,Z 414.998,A -85,B 0,C 180,E1 -8520.268,E2 -8520.268} C_VEL
LIN {X 0,Y 453.513,Z 414.995,A -85,B 0,C 180,E1 -8523.294,E2 -8523.294} C_VEL
LIN {X 0,Y 453.508,Z 414.995,A -85,B 0,C 180,E1 -8526.239,E2 -8526.239} C_VEL
LIN {X 0,Y 453.486,Z 414.998,A -85,B 0,C 180,E1 -8529.118,E2 -8529.118} C_VEL
LIN {X 0,Y 453.514,Z 414.996,A -85,B 0,C 180,E1 -8531.945,E2 -8531.945} C_VEL
LIN {X 0,Y 453.563,Z 415.113,A -85,B 0,C 180,E1 -8534.928,E2 -8534.928} C_VEL
LIN {X 0,Y 456.666,Z 425.801,A -85,B 0,C 180,E1 -8535.631,E2 -8535.631} C_VEL
LIN {X 0,Y 456.504,Z 436.314,A -85,B 0,C 180,E1 -8536.354,E2 -8536.354} C_VEL
LIN {X 0,Y 455.957,Z 447.451,A -85,B 0,C 180,E1 -8537.312,E2 -8537.312} C_VEL
LIN {X 0,Y 455.472,Z 457.806,A -85,B 0,C 180,E1 -8538.428,E2 -8538.428} C_VEL
LIN {X 0,Y 455.248,Z 461.313,A -85,B 0,C 180,E1 -8538.869,E2 -8538.869} C_VEL
LIN {X 0,Y 454.33,Z 465.42,A -85,B 0,C 180,E1 -8539.393,E2 -8539.393} C_VEL
LIN {X 0,Y 451.176,Z 471.828,A -85,B 0,C 180,E1 -8540.264,E2 -8540.264} C_VEL
LIN {X 0,Y 448.041,Z 477.616,A -85,B 0,C 180,E1 -8541.208,E2 -8541.208} C_VEL
LIN {X 0,Y 447.164,Z 480.748,A -85,B 0,C 180,E1 -8541.839,E2 -8541.839} C_VEL
LIN {X 0,Y 446.945,Z 486.257,A -85,B 0,C 180,E1 -8543.227,E2 -8543.227} C_VEL
LIN {X 0,Y 446.522,Z 490.514,A -85,B 0,C 180,E1 -8544.581,E2 -8544.581} C_VEL
LIN {X 0,Y 446.436,Z 492.744,A -85,B 0,C 180,E1 -8545.485,E2 -8545.485} C_VEL
LIN {X 0,Y 446.307,Z 494.568,A -85,B 0,C 180,E1 -8546.389,E2 -8546.389} C_VEL
LIN {X 0,Y 446.18,Z 495.946,A -85,B 0,C 180,E1 -8547.291,E2 -8547.291} C_VEL
LIN {X 0,Y 446.205,Z 496.908,A -85,B 0,C 180,E1 -8548.195,E2 -8548.195} C_VEL
LIN {X 0,Y 446.159,Z 497.739,A -85,B 0,C 180,E1 -8550,E2 -8550} C_VEL
LIN {X 0,Y 446.122,Z 497.563,A -85,B 0,C 180,E1 -8550.903,E2 -8550.903} C_VEL
LIN {X 0,Y 446.204,Z 496.986,A -85,B 0,C 180,E1 -8551.805,E2 -8551.805} C_VEL
LIN {X 0,Y 446.3,Z 494.725,A -85,B 0,C 180,E1 -8553.611,E2 -8553.611} C_VEL
LIN {X 0,Y 446.516,Z 491.919,A -85,B 0,C 180,E1 -8554.966,E2 -8554.966} C_VEL
LIN {X 0,Y 446.846,Z 488.103,A -85,B 0,C 180,E1 -8556.321,E2 -8556.321} C_VEL
LIN {X 0,Y 447.026,Z 482.225,A -85,B 0,C 180,E1 -8557.917,E2 -8557.917} C_VEL
LIN {X 0,Y 447.521,Z 475.813,A -85,B 0,C 180,E1 -8559.263,E2 -8559.263} C_VEL
LIN {X 0,Y 448.06,Z 467.793,A -85,B 0,C 180,E1 -8560.62,E2 -8560.62} C_VEL
LIN {X 0,Y 448.513,Z 459.576,A -85,B 0,C 180,E1 -8561.754,E2 -8561.754} C_VEL
LIN {X 0,Y 449.065,Z 449.397,A -85,B 0,C 180,E1 -8562.886,E2 -8562.886} C_VEL
LIN {X 0,Y 449.598,Z 438.891,A -85,B 0,C 180,E1 -8563.824,E2 -8563.824} C_VEL
LIN {X 0,Y 449.951,Z 428.238,A -85,B 0,C 180,E1 -8564.588,E2 -8564.588} C_VEL
LIN {X 0,Y 446.961,Z 417.622,A -85,B 0,C 180,E1 -8565.322,E2 -8565.322} C_VEL
LIN {X 0,Y 446.517,Z 415.865,A -85,B 0,C 180,E1 -8565.432,E2 -8565.432} C_VEL
LIN {X 0,Y 446.455,Z 415.874,A -85,B 0,C 180,E1 -8568.351,E2 -8568.351} C_VEL
LIN {X 0,Y 446.451,Z 415.875,A -85,B 0,C 180,E1 -8571.755,E2 -8571.755} C_VEL
LIN {X 0,Y 446.462,Z 415.874,A -85,B 0,C 180,E1 -8575.152,E2 -8575.152} C_VEL
LIN {X 0,Y 446.487,Z 415.868,A -85,B 0,C 180,E1 -8578.179,E2 -8578.179} C_VEL
LIN {X 0,Y 446.422,Z 415.877,A -85,B 0,C 180,E1 -8581.775,E2 -8581.775} C_VEL
LIN {X 0,Y 446.433,Z 415.875,A -85,B 0,C 180,E1 -8584.523,E2 -8584.523} C_VEL
LIN {X 0,Y 446.442,Z 415.874,A -85,B 0,C 180,E1 -8588.083,E2 -8588.083} C_VEL
LIN {X 0,Y 446.45,Z 415.876,A -85,B 0,C 180,E1 -8590.921,E2 -8590.921} C_VEL
LIN {X 0,Y 446.448,Z 415.872,A -85,B 0,C 180,E1 -8593.84,E2 -8593.84} C_VEL
LIN {X 0,Y 446.424,Z 415.876,A -85,B 0,C 180,E1 -8596.4,E2 -8596.4} C_VEL
LIN {X 0,Y 446.45,Z 415.873,A -85,B 0,C 180,E1 -8599.803,E2 -8599.803} C_VEL
LIN {X 0,Y 446.412,Z 415.878,A -85,B 0,C 180,E1 -8602.121,E2 -8602.121} C_VEL
LIN {X 0,Y 446.431,Z 415.876,A -85,B 0,C 180,E1 -8605.477,E2 -8605.477} C_VEL
LIN {X 0,Y 446.419,Z 415.88,A -85,B 0,C 180,E1 -8608.7,E2 -8608.7} C_VEL
LIN {X 0,Y 446.487,Z 415.867,A -85,B 0,C 180,E1 -8611.821,E2 -8611.821} C_VEL
LIN {X 0,Y 446.447,Z 415.876,A -85,B 0,C 180,E1 -8614.847,E2 -8614.847} C_VEL
LIN {X 0,Y 446.451,Z 415.875,A -85,B 0,C 180,E1 -8618.245,E2 -8618.245} C_VEL
LIN {X 0,Y 446.461,Z 415.871,A -85,B 0,C 180,E1 -8621.649,E2 -8621.649} C_VEL
LIN {X 0,Y 446.511,Z 415.868,A -85,B 0,C 180,E1 -8624.48,E2 -8624.48} C_VEL
LIN {X 0,Y 446.542,Z 415.863,A -85,B 0,C 180,E1 -8628.194,E2 -8628.194} C_VEL
LIN {X 0,Y 446.537,Z 415.864,A -85,B 0,C 180,E1 -8630.945,E2 -8630.945} C_VEL
LIN {X 0,Y 446.644,Z 415.849,A -85,B 0,C 180,E1 -8633.676,E2 -8633.676} C_VEL
LIN {X 0,Y 446.712,Z 415.84,A -85,B 0,C 180,E1 -8637.295,E2 -8637.295} C_VEL
LIN {X 0,Y 446.797,Z 415.831,A -85,B 0,C 180,E1 -8640,E2 -8640} C_VEL
LIN {X 0,Y 446.713,Z 415.843,A -85,B 0,C 180,E1 -8642.705,E2 -8642.705} C_VEL
LIN {X 0,Y 446.644,Z 415.853,A -85,B 0,C 180,E1 -8646.324,E2 -8646.324} C_VEL
LIN {X 0,Y 446.536,Z 415.862,A -85,B 0,C 180,E1 -8649.055,E2 -8649.055} C_VEL
LIN {X 0,Y 446.537,Z 415.863,A -85,B 0,C 180,E1 -8652.729,E2 -8652.729} C_VEL
LIN {X 0,Y 446.493,Z 415.87,A -85,B 0,C 180,E1 -8656.459,E2 -8656.459} C_VEL
LIN {X 0,Y 446.472,Z 415.87,A -85,B 0,C 180,E1 -8659.303,E2 -8659.303} C_VEL
LIN {X 0,Y 446.42,Z 415.88,A -85,B 0,C 180,E1 -8662.2,E2 -8662.2} C_VEL
LIN {X 0,Y 446.446,Z 415.873,A -85,B 0,C 180,E1 -8665.153,E2 -8665.153} C_VEL
LIN {X 0,Y 446.487,Z 415.871,A -85,B 0,C 180,E1 -8668.179,E2 -8668.179} C_VEL
LIN {X 0,Y 446.423,Z 415.879,A -85,B 0,C 180,E1 -8671.775,E2 -8671.775} C_VEL
LIN {X 0,Y 446.433,Z 415.876,A -85,B 0,C 180,E1 -8674.523,E2 -8674.523} C_VEL
LIN {X 0,Y 446.433,Z 415.878,A -85,B 0,C 180,E1 -8678.082,E2 -8678.082} C_VEL
LIN {X 0,Y 446.43,Z 415.875,A -85,B 0,C 180,E1 -8680.918,E2 -8680.918} C_VEL
LIN {X 0,Y 446.425,Z 415.879,A -85,B 0,C 180,E1 -8683.843,E2 -8683.843} C_VEL
LIN {X 0,Y 446.402,Z 415.882,A -85,B 0,C 180,E1 -8686.403,E2 -8686.403} C_VEL
LIN {X 0,Y 446.491,Z 415.952,A -85,B 0,C 180,E1 -8688.904,E2 -8688.904} C_VEL
LIN {X 0,Y 448.225,Z 424.909,A -85,B 0,C 180,E1 -8691.627,E2 -8691.627} C_VEL
LIN {X 0,Y 449.206,Z 430.494,A -85,B 0,C 180,E1 -8693.243,E2 -8693.243} C_VEL
LIN {X 0,Y 448.786,Z 438.672,A -85,B 0,C 180,E1 -8695.412,E2 -8695.412} C_VEL
LIN {X 0,Y 448.154,Z 452.05,A -85,B 0,C 180,E1 -8698.835,E2 -8698.835} C_VEL
LIN {X 0,Y 447.563,Z 465.435,A -85,B 0,C 180,E1 -8702.15,E2 -8702.15} C_VEL
LIN {X 0,Y 447.062,Z 478.722,A -85,B 0,C 180,E1 -8705.378,E2 -8705.378} C_VEL
LIN {X 0,Y 446.614,Z 492.854,A -85,B 0,C 180,E1 -8708.781,E2 -8708.781} C_VEL
LIN {X 0,Y 446.315,Z 504.726,A -85,B 0,C 180,E1 -8711.643,E2 -8711.643} C_VEL
LIN {X 0,Y 446.094,Z 513.582,A -85,B 0,C 180,E1 -8713.795,E2 -8713.795} C_VEL
LIN {X 0,Y 447.609,Z 528.964,A -85,B 0,C 180,E1 -8714.252,E2 -8714.252} C_VEL
LIN {X 0,Y 448.569,Z 541.291,A -85,B 0,C 180,E1 -8714.786,E2 -8714.786} C_VEL
LIN {X 0,Y 448.639,Z 547.933,A -85,B 0,C 180,E1 -8715.137,E2 -8715.137} C_VEL
LIN {X 0,Y 447.948,Z 560.356,A -85,B 0,C 180,E1 -8715.925,E2 -8715.925} C_VEL
LIN {X 0,Y 447.408,Z 570.845,A -85,B 0,C 180,E1 -8716.774,E2 -8716.774} C_VEL
LIN {X 0,Y 447.011,Z 580.591,A -85,B 0,C 180,E1 -8717.746,E2 -8717.746} C_VEL
LIN {X 0,Y 446.445,Z 589.924,A -85,B 0,C 180,E1 -8718.881,E2 -8718.881} C_VEL
LIN {X 0,Y 446.055,Z 599.061,A -85,B 0,C 180,E1 -8720.249,E2 -8720.249} C_VEL
LIN {X 0,Y 445.858,Z 606.448,A -85,B 0,C 180,E1 -8721.616,E2 -8721.616} C_VEL
LIN {X 0,Y 445.776,Z 611.449,A -85,B 0,C 180,E1 -8722.754,E2 -8722.754} C_VEL
LIN {X 0,Y 445.786,Z 616.327,A -85,B 0,C 180,E1 -8724.118,E2 -8724.118} C_VEL
LIN {X 0,Y 445.812,Z 620.06,A -85,B 0,C 180,E1 -8725.479,E2 -8725.479} C_VEL
LIN {X 0,Y 445.831,Z 621.987,A -85,B 0,C 180,E1 -8726.385,E2 -8726.385} C_VEL
LIN {X 0,Y 445.823,Z 623.43,A -85,B 0,C 180,E1 -8727.289,E2 -8727.289} C_VEL
LIN {X 0,Y 445.819,Z 624.459,A -85,B 0,C 180,E1 -8728.193,E2 -8728.193} C_VEL
LIN {X 0,Y 445.968,Z 625.333,A -85,B 0,C 180,E1 -8730,E2 -8730} C_VEL
LIN {X 0,Y 445.819,Z 624.461,A -85,B 0,C 180,E1 -8731.807,E2 -8731.807} C_VEL
LIN {X 0,Y 445.823,Z 623.433,A -85,B 0,C 180,E1 -8732.711,E2 -8732.711} C_VEL
LIN {X 0,Y 445.831,Z 621.989,A -85,B 0,C 180,E1 -8733.615,E2 -8733.615} C_VEL
LIN {X 0,Y 445.81,Z 618.953,A -85,B 0,C 180,E1 -8734.974,E2 -8734.974} C_VEL
LIN {X 0,Y 445.758,Z 613.74,A -85,B 0,C 180,E1 -8736.643,E2 -8736.643} C_VEL
LIN {X 0,Y 445.861,Z 607.505,A -85,B 0,C 180,E1 -8738.156,E2 -8738.156} C_VEL
LIN {X 0,Y 446.036,Z 600.418,A -85,B 0,C 180,E1 -8739.523,E2 -8739.523} C_VEL
LIN {X 0,Y 446.369,Z 591.581,A -85,B 0,C 180,E1 -8740.891,E2 -8740.891} C_VEL
LIN {X 0,Y 446.832,Z 582.56,A -85,B 0,C 180,E1 -8742.029,E2 -8742.029} C_VEL
LIN {X 0,Y 447.307,Z 571.973,A -85,B 0,C 180,E1 -8743.121,E2 -8743.121} C_VEL
LIN {X 0,Y 447.862,Z 561.901,A -85,B 0,C 180,E1 -8743.962,E2 -8743.962} C_VEL
LIN {X 0,Y 448.513,Z 549.9,A -85,B 0,C 180,E1 -8744.752,E2 -8744.752} C_VEL
LIN {X 0,Y 448.703,Z 542.412,A -85,B 0,C 180,E1 -8745.152,E2 -8745.152} C_VEL
LIN {X 0,Y 447.767,Z 530.864,A -85,B 0,C 180,E1 -8745.673,E2 -8745.673} C_VEL
LIN {X 0,Y 446.535,Z 517.889,A -85,B 0,C 180,E1 -8746.092,E2 -8746.092} C_VEL
LIN {X 0,Y 446.082,Z 513.649,A -85,B 0,C 180,E1 -8746.19,E2 -8746.19} C_VEL
LIN {X 0,Y 446.402,Z 500.788,A -85,B 0,C 180,E1 -8749.306,E2 -8749.306} C_VEL
LIN {X 0,Y 446.843,Z 485.819,A -85,B 0,C 180,E1 -8752.909,E2 -8752.909} C_VEL
LIN {X 0,Y 447.285,Z 472.599,A -85,B 0,C 180,E1 -8756.101,E2 -8756.101} C_VEL
LIN {X 0,Y 447.811,Z 459.234,A -85,B 0,C 180,E1 -8759.37,E2 -8759.37} C_VEL
LIN {X 0,Y 448.38,Z 446.873,A -85,B 0,C 180,E1 -8762.469,E2 -8762.469} C_VEL
LIN {X 0,Y 449.169,Z 433.473,A -85,B 0,C 180,E1 -8765.943,E2 -8765.943} C_VEL
LIN {X 0,Y 449.072,Z 429.445,A -85,B 0,C 180,E1 -8767.046,E2 -8767.046} C_VEL
LIN {X 0,Y 447.131,Z 419.044,A -85,B 0,C 180,E1 -8770.124,E2 -8770.124} C_VEL
LIN {X 0,Y 446.472,Z 415.874,A -85,B 0,C 180,E1 -8771.119,E2 -8771.119} C_VEL
LIN {X 0,Y 446.457,Z 415.874,A -85,B 0,C 180,E1 -8774.897,E2 -8774.897} C_VEL
LIN {X 0,Y 446.439,Z 415.877,A -85,B 0,C 180,E1 -8777.722,E2 -8777.722} C_VEL
LIN {X 0,Y 446.46,Z 415.871,A -85,B 0,C 180,E1 -8780.974,E2 -8780.974} C_VEL
LIN {X 0,Y 446.424,Z 415.878,A -85,B 0,C 180,E1 -8784.374,E2 -8784.374} C_VEL
LIN {X 0,Y 446.426,Z 415.879,A -85,B 0,C 180,E1 -8787.639,E2 -8787.639} C_VEL
LIN {X 0,Y 446.453,Z 415.872,A -85,B 0,C 180,E1 -8790.791,E2 -8790.791} C_VEL
LIN {X 0,Y 446.481,Z 415.872,A -85,B 0,C 180,E1 -8793.849,E2 -8793.849} C_VEL
LIN {X 0,Y 446.43,Z 415.875,A -85,B 0,C 180,E1 -8796.823,E2 -8796.823} C_VEL
LIN {X 0,Y 446.449,Z 415.876,A -85,B 0,C 180,E1 -8799.737,E2 -8799.737} C_VEL
LIN {X 0,Y 446.468,Z 415.871,A -85,B 0,C 180,E1 -8802.597,E2 -8802.597} C_VEL
LIN {X 0,Y 446.474,Z 415.872,A -85,B 0,C 180,E1 -8805.413,E2 -8805.413} C_VEL
LIN {X 0,Y 446.543,Z 415.863,A -85,B 0,C 180,E1 -8808.194,E2 -8808.194} C_VEL
LIN {X 0,Y 446.537,Z 415.862,A -85,B 0,C 180,E1 -8810.945,E2 -8810.945} C_VEL
LIN {X 0,Y 446.645,Z 415.852,A -85,B 0,C 180,E1 -8813.676,E2 -8813.676} C_VEL
LIN {X 0,Y 446.714,Z 415.843,A -85,B 0,C 180,E1 -8817.295,E2 -8817.295} C_VEL
LIN {X 0,Y 446.798,Z 415.831,A -85,B 0,C 180,E1 -8820,E2 -8820} C_VEL
LIN {X 0,Y 446.696,Z 415.841,A -85,B 0,C 180,E1 -8822.705,E2 -8822.705} C_VEL
LIN {X 0,Y 446.641,Z 415.849,A -85,B 0,C 180,E1 -8826.324,E2 -8826.324} C_VEL
LIN {X 0,Y 446.538,Z 415.864,A -85,B 0,C 180,E1 -8829.055,E2 -8829.055} C_VEL
LIN {X 0,Y 446.538,Z 415.862,A -85,B 0,C 180,E1 -8832.729,E2 -8832.729} C_VEL
LIN {X 0,Y 446.494,Z 415.866,A -85,B 0,C 180,E1 -8836.459,E2 -8836.459} C_VEL
LIN {X 0,Y 446.474,Z 415.874,A -85,B 0,C 180,E1 -8839.303,E2 -8839.303} C_VEL
LIN {X 0,Y 446.422,Z 415.876,A -85,B 0,C 180,E1 -8842.2,E2 -8842.2} C_VEL
LIN {X 0,Y 446.461,Z 415.874,A -85,B 0,C 180,E1 -8845.152,E2 -8845.152} C_VEL
LIN {X 0,Y 446.488,Z 415.867,A -85,B 0,C 180,E1 -8848.179,E2 -8848.179} C_VEL
LIN {X 0,Y 446.424,Z 415.877,A -85,B 0,C 180,E1 -8851.775,E2 -8851.775} C_VEL
LIN {X 0,Y 446.432,Z 415.876,A -85,B 0,C 180,E1 -8854.523,E2 -8854.523} C_VEL
LIN {X 0,Y 446.418,Z 415.877,A -85,B 0,C 180,E1 -8858.079,E2 -8858.079} C_VEL
LIN {X 0,Y 446.431,Z 415.878,A -85,B 0,C 180,E1 -8860.918,E2 -8860.918} C_VEL
LIN {X 0,Y 446.426,Z 415.875,A -85,B 0,C 180,E1 -8863.843,E2 -8863.843} C_VEL
LIN {X 0,Y 446.451,Z 415.873,A -85,B 0,C 180,E1 -8866.397,E2 -8866.397} C_VEL
LIN {X 0,Y 446.473,Z 415.87,A -85,B 0,C 180,E1 -8869.805,E2 -8869.805} C_VEL
LIN {X 0,Y 446.437,Z 415.874,A -85,B 0,C 180,E1 -8872.124,E2 -8872.124} C_VEL
LIN {X 0,Y 446.432,Z 415.876,A -85,B 0,C 180,E1 -8875.477,E2 -8875.477} C_VEL
LIN {X 0,Y 446.42,Z 415.88,A -85,B 0,C 180,E1 -8878.7,E2 -8878.7} C_VEL
LIN {X 0,Y 446.488,Z 415.867,A -85,B 0,C 180,E1 -8881.821,E2 -8881.821} C_VEL
LIN {X 0,Y 446.462,Z 415.875,A -85,B 0,C 180,E1 -8884.848,E2 -8884.848} C_VEL
LIN {X 0,Y 446.452,Z 415.874,A -85,B 0,C 180,E1 -8888.245,E2 -8888.245} C_VEL
LIN {X 0,Y 446.46,Z 415.873,A -85,B 0,C 180,E1 -8891.649,E2 -8891.649} C_VEL
LIN {X 0,Y 446.504,Z 415.869,A -85,B 0,C 180,E1 -8894.655,E2 -8894.655} C_VEL
LIN {X 0,Y 449.7,Z 426.838,A -85,B 0,C 180,E1 -8895.404,E2 -8895.404} C_VEL
LIN {X 0,Y 449.944,Z 429.876,A -85,B 0,C 180,E1 -8895.614,E2 -8895.614} C_VEL
LIN {X 0,Y 449.446,Z 440.976,A -85,B 0,C 180,E1 -8896.434,E2 -8896.434} C_VEL
LIN {X 0,Y 448.915,Z 451.829,A -85,B 0,C 180,E1 -8897.454,E2 -8897.454} C_VEL
LIN {X 0,Y 448.356,Z 462.355,A -85,B 0,C 180,E1 -8898.7,E2 -8898.7} C_VEL
LIN {X 0,Y 447.896,Z 470.107,A -85,B 0,C 180,E1 -8899.832,E2 -8899.832} C_VEL
LIN {X 0,Y 447.368,Z 477.685,A -85,B 0,C 180,E1 -8901.189,E2 -8901.189} C_VEL
LIN {X 0,Y 447.164,Z 480.748,A -85,B 0,C 180,E1 -8901.839,E2 -8901.839} C_VEL
LIN {X 0,Y 446.299,Z 483.671,A -85,B 0,C 180,E1 -8902.49,E2 -8902.49} C_VEL
LIN {X 0,Y 443.227,Z 488.126,A -85,B 0,C 180,E1 -8903.562,E2 -8903.562} C_VEL
LIN {X 0,Y 440.205,Z 491.913,A -85,B 0,C 180,E1 -8904.686,E2 -8904.686} C_VEL
LIN {X 0,Y 439.43,Z 493.743,A -85,B 0,C 180,E1 -8905.41,E2 -8905.41} C_VEL
LIN {X 0,Y 439.293,Z 495.574,A -85,B 0,C 180,E1 -8906.331,E2 -8906.331} C_VEL
LIN {X 0,Y 439.16,Z 496.952,A -85,B 0,C 180,E1 -8907.248,E2 -8907.248} C_VEL
LIN {X 0,Y 439.184,Z 497.913,A -85,B 0,C 180,E1 -8908.166,E2 -8908.166} C_VEL
LIN {X 0,Y 439.152,Z 498.741,A -85,B 0,C 180,E1 -8910,E2 -8910} C_VEL
LIN {X 0,Y 439.099,Z 498.567,A -85,B 0,C 180,E1 -8910.917,E2 -8910.917} C_VEL
LIN {X 0,Y 439.184,Z 497.99,A -85,B 0,C 180,E1 -8911.834,E2 -8911.834} C_VEL
LIN {X 0,Y 439.286,Z 495.73,A -85,B 0,C 180,E1 -8913.669,E2 -8913.669} C_VEL
LIN {X 0,Y 439.516,Z 492.922,A -85,B 0,C 180,E1 -8915.045,E2 -8915.045} C_VEL
LIN {X 0,Y 439.868,Z 489.106,A -85,B 0,C 180,E1 -8916.421,E2 -8916.421} C_VEL
LIN {X 0,Y 440.066,Z 483.229,A -85,B 0,C 180,E1 -8918.042,E2 -8918.042} C_VEL
LIN {X 0,Y 440.588,Z 476.816,A -85,B 0,C 180,E1 -8919.41,E2 -8919.41} C_VEL
LIN {X 0,Y 441.157,Z 468.795,A -85,B 0,C 180,E1 -8920.789,E2 -8920.789} C_VEL
LIN {X 0,Y 441.635,Z 460.577,A -85,B 0,C 180,E1 -8921.939,E2 -8921.939} C_VEL
LIN {X 0,Y 442.216,Z 450.398,A -85,B 0,C 180,E1 -8923.089,E2 -8923.089} C_VEL
LIN {X 0,Y 442.777,Z 439.891,A -85,B 0,C 180,E1 -8924.042,E2 -8924.042} C_VEL
LIN {X 0,Y 443.064,Z 429.249,A -85,B 0,C 180,E1 -8924.82,E2 -8924.82} C_VEL
LIN {X 0,Y 439.564,Z 417.335,A -85,B 0,C 180,E1 -8925.653,E2 -8925.653} C_VEL
LIN {X 0,Y 439.471,Z 416.743,A -85,B 0,C 180,E1 -8925.716,E2 -8925.716} C_VEL
LIN {X 0,Y 439.444,Z 416.749,A -85,B 0,C 180,E1 -8929.337,E2 -8929.337} C_VEL
LIN {X 0,Y 439.369,Z 416.755,A -85,B 0,C 180,E1 -8932.575,E2 -8932.575} C_VEL
LIN {X 0,Y 439.409,Z 416.752,A -85,B 0,C 180,E1 -8935.585,E2 -8935.585} C_VEL
LIN {X 0,Y 439.42,Z 416.749,A -85,B 0,C 180,E1 -8938.673,E2 -8938.673} C_VEL
LIN {X 0,Y 439.373,Z 416.753,A -85,B 0,C 180,E1 -8942.03,E2 -8942.03} C_VEL
LIN {X 0,Y 439.399,Z 416.754,A -85,B 0,C 180,E1 -8945.341,E2 -8945.341} C_VEL
LIN {X 0,Y 439.402,Z 416.752,A -85,B 0,C 180,E1 -8948.593,E2 -8948.593} C_VEL
LIN {X 0,Y 439.408,Z 416.753,A -85,B 0,C 180,E1 -8951.259,E2 -8951.259} C_VEL
LIN {X 0,Y 439.412,Z 416.753,A -85,B 0,C 180,E1 -8954.728,E2 -8954.728} C_VEL
LIN {X 0,Y 439.4,Z 416.75,A -85,B 0,C 180,E1 -8957.796,E2 -8957.796} C_VEL
LIN {X 0,Y 439.432,Z 416.747,A -85,B 0,C 180,E1 -8960.228,E2 -8960.228} C_VEL
LIN {X 0,Y 439.376,Z 416.754,A -85,B 0,C 180,E1 -8963.713,E2 -8963.713} C_VEL
LIN {X 0,Y 439.375,Z 416.757,A -85,B 0,C 180,E1 -8967.054,E2 -8967.054} C_VEL
LIN {X 0,Y 439.385,Z 416.753,A -85,B 0,C 180,E1 -8970.274,E2 -8970.274} C_VEL
LIN {X 0,Y 439.432,Z 416.747,A -85,B 0,C 180,E1 -8973.396,E2 -8973.396} C_VEL
LIN {X 0,Y 439.387,Z 416.755,A -85,B 0,C 180,E1 -8976.429,E2 -8976.429} C_VEL
LIN {X 0,Y 439.392,Z 416.752,A -85,B 0,C 180,E1 -8979.397,E2 -8979.397} C_VEL
LIN {X 0,Y 439.435,Z 416.749,A -85,B 0,C 180,E1 -8982.31,E2 -8982.31} C_VEL
LIN {X 0,Y 439.451,Z 416.745,A -85,B 0,C 180,E1 -8985.174,E2 -8985.174} C_VEL
LIN {X 0,Y 439.511,Z 416.738,A -85,B 0,C 180,E1 -8988.002,E2 -8988.002} C_VEL
LIN {X 0,Y 439.507,Z 416.738,A -85,B 0,C 180,E1 -8991.725,E2 -8991.725} C_VEL
LIN {X 0,Y 439.623,Z 416.727,A -85,B 0,C 180,E1 -8994.496,E2 -8994.496} C_VEL
LIN {X 0,Y 439.639,Z 416.725,A -85,B 0,C 180,E1 -8998.168,E2 -8998.168} C_VEL
LIN {X 0,Y 439.767,Z 416.707,A -85,B 0,C 180,E1 -9000,E2 -9000} C_VEL
LIN {X 0,Y 439.66,Z 416.721,A -85,B 0,C 180,E1 -9002.749,E2 -9002.749} C_VEL
LIN {X 0,Y 439.616,Z 416.727,A -85,B 0,C 180,E1 -9006.425,E2 -9006.425} C_VEL
LIN {X 0,Y 439.499,Z 416.738,A -85,B 0,C 180,E1 -9009.202,E2 -9009.202} C_VEL
LIN {X 0,Y 439.507,Z 416.738,A -85,B 0,C 180,E1 -9012.726,E2 -9012.726} C_VEL
LIN {X 0,Y 439.45,Z 416.748,A -85,B 0,C 180,E1 -9016.349,E2 -9016.349} C_VEL
LIN {X 0,Y 439.405,Z 416.752,A -85,B 0,C 180,E1 -9019.626,E2 -9019.626} C_VEL
LIN {X 0,Y 439.366,Z 416.757,A -85,B 0,C 180,E1 -9022.575,E2 -9022.575} C_VEL
LIN {X 0,Y 439.4,Z 416.752,A -85,B 0,C 180,E1 -9025.585,E2 -9025.585} C_VEL
LIN {X 0,Y 439.42,Z 416.748,A -85,B 0,C 180,E1 -9028.673,E2 -9028.673} C_VEL
LIN {X 0,Y 439.373,Z 416.757,A -85,B 0,C 180,E1 -9032.031,E2 -9032.031} C_VEL
LIN {X 0,Y 439.398,Z 416.752,A -85,B 0,C 180,E1 -9035.341,E2 -9035.341} C_VEL
LIN {X 0,Y 439.391,Z 416.752,A -85,B 0,C 180,E1 -9038.594,E2 -9038.594} C_VEL
LIN {X 0,Y 439.391,Z 416.752,A -85,B 0,C 180,E1 -9041.257,E2 -9041.257} C_VEL
LIN {X 0,Y 439.407,Z 416.756,A -85,B 0,C 180,E1 -9044.729,E2 -9044.729} C_VEL
LIN {X 0,Y 439.438,Z 416.849,A -85,B 0,C 180,E1 -9048.596,E2 -9048.596} C_VEL
LIN {X 0,Y 441.349,Z 426.573,A -85,B 0,C 180,E1 -9051.608,E2 -9051.608} C_VEL
LIN {X 0,Y 442.312,Z 432.803,A -85,B 0,C 180,E1 -9053.427,E2 -9053.427} C_VEL
LIN {X 0,Y 441.513,Z 446.095,A -85,B 0,C 180,E1 -9056.962,E2 -9056.962} C_VEL
LIN {X 0,Y 440.876,Z 458.439,A -85,B 0,C 180,E1 -9060.128,E2 -9060.128} C_VEL
LIN {X 0,Y 440.343,Z 471.318,A -85,B 0,C 180,E1 -9063.352,E2 -9063.352} C_VEL
LIN {X 0,Y 439.795,Z 485.911,A -85,B 0,C 180,E1 -9066.951,E2 -9066.951} C_VEL
LIN {X 0,Y 439.366,Z 499.836,A -85,B 0,C 180,E1 -9070.372,E2 -9070.372} C_VEL
LIN {X 0,Y 439.021,Z 512.588,A -85,B 0,C 180,E1 -9073.533,E2 -9073.533} C_VEL
LIN {X 0,Y 440.53,Z 527.398,A -85,B 0,C 180,E1 -9073.975,E2 -9073.975} C_VEL
LIN {X 0,Y 441.467,Z 540.244,A -85,B 0,C 180,E1 -9074.535,E2 -9074.535} C_VEL
LIN {X 0,Y 441.751,Z 546.918,A -85,B 0,C 180,E1 -9074.899,E2 -9074.899} C_VEL
LIN {X 0,Y 440.991,Z 559.333,A -85,B 0,C 180,E1 -9075.699,E2 -9075.699} C_VEL
LIN {X 0,Y 440.408,Z 570.09,A -85,B 0,C 180,E1 -9076.585,E2 -9076.585} C_VEL
LIN {X 0,Y 440.027,Z 579.57,A -85,B 0,C 180,E1 -9077.548,E2 -9077.548} C_VEL
LIN {X 0,Y 439.426,Z 588.903,A -85,B 0,C 180,E1 -9078.701,E2 -9078.701} C_VEL
LIN {X 0,Y 438.995,Z 598.038,A -85,B 0,C 180,E1 -9080.09,E2 -9080.09} C_VEL
LIN {X 0,Y 438.795,Z 605.428,A -85,B 0,C 180,E1 -9081.48,E2 -9081.48} C_VEL
LIN {X 0,Y 438.707,Z 610.431,A -85,B 0,C 180,E1 -9082.637,E2 -9082.637} C_VEL
LIN {X 0,Y 438.725,Z 615.312,A -85,B 0,C 180,E1 -9084.023,E2 -9084.023} C_VEL
LIN {X 0,Y 438.767,Z 619.049,A -85,B 0,C 180,E1 -9085.406,E2 -9085.406} C_VEL
LIN {X 0,Y 438.79,Z 620.978,A -85,B 0,C 180,E1 -9086.327,E2 -9086.327} C_VEL
LIN {X 0,Y 438.781,Z 622.422,A -85,B 0,C 180,E1 -9087.246,E2 -9087.246} C_VEL
LIN {X 0,Y 438.783,Z 623.453,A -85,B 0,C 180,E1 -9088.164,E2 -9088.164} C_VEL
LIN {X 0,Y 438.948,Z 624.329,A -85,B 0,C 180,E1 -9090,E2 -9090} C_VEL
LIN {X 0,Y 438.783,Z 623.454,A -85,B 0,C 180,E1 -9091.836,E2 -9091.836} C_VEL
LIN {X 0,Y 438.781,Z 622.424,A -85,B 0,C 180,E1 -9092.754,E2 -9092.754} C_VEL
LIN {X 0,Y 438.79,Z 620.98,A -85,B 0,C 180,E1 -9093.673,E2 -9093.673} C_VEL
LIN {X 0,Y 438.761,Z 617.941,A -85,B 0,C 180,E1 -9095.054,E2 -9095.054} C_VEL
LIN {X 0,Y 438.686,Z 613.095,A -85,B 0,C 180,E1 -9096.647,E2 -9096.647} C_VEL
LIN {X 0,Y 438.777,Z 606.481,A -85,B 0,C 180,E1 -9098.288,E2 -9098.288} C_VEL
LIN {X 0,Y 438.969,Z 599.392,A -85,B 0,C 180,E1 -9099.678,E2 -9099.678} C_VEL
LIN {X 0,Y 439.334,Z 590.554,A -85,B 0,C 180,E1 -9101.068,E2 -9101.068} C_VEL
LIN {X 0,Y 439.863,Z 581.538,A -85,B 0,C 180,E1 -9102.222,E2 -9102.222} C_VEL
LIN {X 0,Y 440.284,Z 571.825,A -85,B 0,C 180,E1 -9103.248,E2 -9103.248} C_VEL
LIN {X 0,Y 440.921,Z 560.874,A -85,B 0,C 180,E1 -9104.186,E2 -9104.186} C_VEL
LIN {X 0,Y 441.629,Z 548.877,A -85,B 0,C 180,E1 -9104.987,E2 -9104.987} C_VEL
LIN {X 0,Y 441.681,Z 542.513,A -85,B 0,C 180,E1 -9105.34,E2 -9105.34} C_VEL
LIN {X 0,Y 440.733,Z 530.049,A -85,B 0,C 180,E1 -9105.92,E2 -9105.92} C_VEL
LIN {X 0,Y 439.472,Z 516.795,A -85,B 0,C 180,E1 -9106.359,E2 -9106.359} C_VEL
LIN {X 0,Y 439.028,Z 512.565,A -85,B 0,C 180,E1 -9106.467,E2 -9106.467} C_VEL
LIN {X 0,Y 439.361,Z 499.818,A -85,B 0,C 180,E1 -9109.628,E2 -9109.628} C_VEL
LIN {X 0,Y 439.809,Z 484.892,A -85,B 0,C 180,E1 -9113.297,E2 -9113.297} C_VEL
LIN {X 0,Y 440.316,Z 471.332,A -85,B 0,C 180,E1 -9116.641,E2 -9116.641} C_VEL
LIN {X 0,Y 440.876,Z 458.416,A -85,B 0,C 180,E1 -9119.871,E2 -9119.871} C_VEL
LIN {X 0,Y 441.509,Z 446.064,A -85,B 0,C 180,E1 -9123.038,E2 -9123.038} C_VEL
LIN {X 0,Y 442.306,Z 432.765,A -85,B 0,C 180,E1 -9126.574,E2 -9126.574} C_VEL
LIN {X 0,Y 441.142,Z 425.574,A -85,B 0,C 180,E1 -9128.681,E2 -9128.681} C_VEL
LIN {X 0,Y 439.422,Z 416.749,A -85,B 0,C 180,E1 -9131.438,E2 -9131.438} C_VEL
LIN {X 0,Y 439.408,Z 416.751,A -85,B 0,C 180,E1 -9135.271,E2 -9135.271} C_VEL
LIN {X 0,Y 439.393,Z 416.757,A -85,B 0,C 180,E1 -9138.743,E2 -9138.743} C_VEL
LIN {X 0,Y 439.388,Z 416.754,A -85,B 0,C 180,E1 -9141.606,E2 -9141.606} C_VEL
LIN {X 0,Y 439.404,Z 416.75,A -85,B 0,C 180,E1 -9144.844,E2 -9144.844} C_VEL
LIN {X 0,Y 439.377,Z 416.758,A -85,B 0,C 180,E1 -9148.14,E2 -9148.14} C_VEL
LIN {X 0,Y 439.436,Z 416.748,A -85,B 0,C 180,E1 -9151.598,E2 -9151.598} C_VEL
LIN {X 0,Y 439.401,Z 416.752,A -85,B 0,C 180,E1 -9154.415,E2 -9154.415} C_VEL
LIN {X 0,Y 439.367,Z 416.756,A -85,B 0,C 180,E1 -9157.425,E2 -9157.425} C_VEL
LIN {X 0,Y 439.445,Z 416.745,A -85,B 0,C 180,E1 -9160.663,E2 -9160.663} C_VEL
LIN {X 0,Y 439.466,Z 416.744,A -85,B 0,C 180,E1 -9164.225,E2 -9164.225} C_VEL
LIN {X 0,Y 439.511,Z 416.74,A -85,B 0,C 180,E1 -9168.002,E2 -9168.002} C_VEL
LIN {X 0,Y 439.507,Z 416.741,A -85,B 0,C 180,E1 -9171.726,E2 -9171.726} C_VEL
LIN {X 0,Y 439.624,Z 416.723,A -85,B 0,C 180,E1 -9174.496,E2 -9174.496} C_VEL
LIN {X 0,Y 439.641,Z 416.722,A -85,B 0,C 180,E1 -9178.168,E2 -9178.168} C_VEL
LIN {X 0,Y 439.768,Z 416.707,A -85,B 0,C 180,E1 -9180,E2 -9180} C_VEL
LIN {X 0,Y 439.645,Z 416.72,A -85,B 0,C 180,E1 -9182.749,E2 -9182.749} C_VEL
LIN {X 0,Y 439.614,Z 416.724,A -85,B 0,C 180,E1 -9186.425,E2 -9186.425} C_VEL
LIN {X 0,Y 439.501,Z 416.741,A -85,B 0,C 180,E1 -9189.202,E2 -9189.202} C_VEL
LIN {X 0,Y 439.508,Z 416.737,A -85,B 0,C 180,E1 -9192.727,E2 -9192.727} C_VEL
LIN {X 0,Y 439.451,Z 416.743,A -85,B 0,C 180,E1 -9196.349,E2 -9196.349} C_VEL
LIN {X 0,Y 439.407,Z 416.753,A -85,B 0,C 180,E1 -9199.626,E2 -9199.626} C_VEL
LIN {X 0,Y 439.369,Z 416.755,A -85,B 0,C 180,E1 -9202.575,E2 -9202.575} C_VEL
LIN {X 0,Y 439.409,Z 416.752,A -85,B 0,C 180,E1 -9205.585,E2 -9205.585} C_VEL
LIN {X 0,Y 439.421,Z 416.749,A -85,B 0,C 180,E1 -9208.673,E2 -9208.673} C_VEL
LIN {X 0,Y 439.374,Z 416.754,A -85,B 0,C 180,E1 -9212.031,E2 -9212.031} C_VEL
LIN {X 0,Y 439.398,Z 416.754,A -85,B 0,C 180,E1 -9215.34,E2 -9215.34} C_VEL
LIN {X 0,Y 439.38,Z 416.755,A -85,B 0,C 180,E1 -9218.595,E2 -9218.595} C_VEL
LIN {X 0,Y 439.393,Z 416.756,A -85,B 0,C 180,E1 -9221.257,E2 -9221.257} C_VEL
LIN {X 0,Y 439.41,Z 416.752,A -85,B 0,C 180,E1 -9224.728,E2 -9224.728} C_VEL
LIN {X 0,Y 439.416,Z 416.749,A -85,B 0,C 180,E1 -9227.798,E2 -9227.798} C_VEL
LIN {X 0,Y 439.456,Z 416.744,A -85,B 0,C 180,E1 -9230.23,E2 -9230.23} C_VEL
LIN {X 0,Y 439.379,Z 416.753,A -85,B 0,C 180,E1 -9233.713,E2 -9233.713} C_VEL
LIN {X 0,Y 439.376,Z 416.758,A -85,B 0,C 180,E1 -9237.054,E2 -9237.054} C_VEL
LIN {X 0,Y 439.386,Z 416.753,A -85,B 0,C 180,E1 -9240.274,E2 -9240.274} C_VEL
LIN {X 0,Y 439.433,Z 416.748,A -85,B 0,C 180,E1 -9243.396,E2 -9243.396} C_VEL
LIN {X 0,Y 439.391,Z 416.754,A -85,B 0,C 180,E1 -9246.43,E2 -9246.43} C_VEL
LIN {X 0,Y 439.392,Z 416.752,A -85,B 0,C 180,E1 -9249.397,E2 -9249.397} C_VEL
LIN {X 0,Y 439.434,Z 416.75,A -85,B 0,C 180,E1 -9252.309,E2 -9252.309} C_VEL
LIN {X 0,Y 439.491,Z 416.9,A -85,B 0,C 180,E1 -9254.419,E2 -9254.419} C_VEL
LIN {X 0,Y 442.738,Z 427.875,A -85,B 0,C 180,E1 -9255.169,E2 -9255.169} C_VEL
LIN {X 0,Y 443.148,Z 430.99,A -85,B 0,C 180,E1 -9255.396,E2 -9255.396} C_VEL
LIN {X 0,Y 442.621,Z 441.986,A -85,B 0,C 180,E1 -9256.221,E2 -9256.221} C_VEL
LIN {X 0,Y 442.058,Z 452.839,A -85,B 0,C 180,E1 -9257.256,E2 -9257.256} C_VEL
LIN {X 0,Y 441.47,Z 463.363,A -85,B 0,C 180,E1 -9258.522,E2 -9258.522} C_VEL
LIN {X 0,Y 440.983,Z 471.114,A -85,B 0,C 180,E1 -9259.671,E2 -9259.671} C_VEL
LIN {X 0,Y 440.425,Z 478.692,A -85,B 0,C 180,E1 -9261.049,E2 -9261.049} C_VEL
LIN {X 0,Y 440.137,Z 483.972,A -85,B 0,C 180,E1 -9262.233,E2 -9262.233} C_VEL
LIN {X 0,Y 439.885,Z 488.819,A -85,B 0,C 180,E1 -9263.579,E2 -9263.579} C_VEL
LIN {X 0,Y 439.523,Z 492.708,A -85,B 0,C 180,E1 -9264.954,E2 -9264.954} C_VEL
LIN {X 0,Y 439.43,Z 493.743,A -85,B 0,C 180,E1 -9265.41,E2 -9265.41} C_VEL
LIN {X 0,Y 438.651,Z 495.37,A -85,B 0,C 180,E1 -9266.145,E2 -9266.145} C_VEL
LIN {X 0,Y 435.652,Z 497.663,A -85,B 0,C 180,E1 -9267.349,E2 -9267.349} C_VEL
LIN {X 0,Y 432.73,Z 499.192,A -85,B 0,C 180,E1 -9268.585,E2 -9268.585} C_VEL
LIN {X 0,Y 432.084,Z 499.594,A -85,B 0,C 180,E1 -9269.362,E2 -9269.362} C_VEL
LIN {X 0,Y 432.075,Z 499.572,A -85,B 0,C 180,E1 -9270.932,E2 -9270.932} C_VEL
LIN {X 0,Y 432.163,Z 498.994,A -85,B 0,C 180,E1 -9271.864,E2 -9271.864} C_VEL
LIN {X 0,Y 432.272,Z 496.734,A -85,B 0,C 180,E1 -9273.729,E2 -9273.729} C_VEL
LIN {X 0,Y 432.517,Z 493.926,A -85,B 0,C 180,E1 -9275.127,E2 -9275.127} C_VEL
LIN {X 0,Y 432.889,Z 490.109,A -85,B 0,C 180,E1 -9276.525,E2 -9276.525} C_VEL
LIN {X 0,Y 433.108,Z 484.234,A -85,B 0,C 180,E1 -9278.172,E2 -9278.172} C_VEL
LIN {X 0,Y 433.659,Z 477.818,A -85,B 0,C 180,E1 -9279.562,E2 -9279.562} C_VEL
LIN {X 0,Y 434.258,Z 469.797,A -85,B 0,C 180,E1 -9280.962,E2 -9280.962} C_VEL
LIN {X 0,Y 434.762,Z 461.579,A -85,B 0,C 180,E1 -9282.131,E2 -9282.131} C_VEL
LIN {X 0,Y 435.374,Z 451.398,A -85,B 0,C 180,E1 -9283.299,E2 -9283.299} C_VEL
LIN {X 0,Y 435.962,Z 440.893,A -85,B 0,C 180,E1 -9284.265,E2 -9284.265} C_VEL
LIN {X 0,Y 436.315,Z 431.973,A -85,B 0,C 180,E1 -9284.935,E2 -9284.935} C_VEL
LIN {X 0,Y 435.076,Z 426.665,A -85,B 0,C 180,E1 -9285.338,E2 -9285.338} C_VEL
LIN {X 0,Y 432.42,Z 417.622,A -85,B 0,C 180,E1 -9285.979,E2 -9285.979} C_VEL
LIN {X 0,Y 432.389,Z 417.627,A -85,B 0,C 180,E1 -9289.485,E2 -9289.485} C_VEL
LIN {X 0,Y 432.323,Z 417.634,A -85,B 0,C 180,E1 -9292.964,E2 -9292.964} C_VEL
LIN {X 0,Y 432.368,Z 417.627,A -85,B 0,C 180,E1 -9296.032,E2 -9296.032} C_VEL
LIN {X 0,Y 432.346,Z 417.633,A -85,B 0,C 180,E1 -9299.187,E2 -9299.187} C_VEL
LIN {X 0,Y 432.326,Z 417.631,A -85,B 0,C 180,E1 -9302.443,E2 -9302.443} C_VEL
LIN {X 0,Y 432.349,Z 417.631,A -85,B 0,C 180,E1 -9305.632,E2 -9305.632} C_VEL
LIN {X 0,Y 432.364,Z 417.629,A -85,B 0,C 180,E1 -9308.718,E2 -9308.718} C_VEL
LIN {X 0,Y 432.377,Z 417.625,A -85,B 0,C 180,E1 -9311.792,E2 -9311.792} C_VEL
LIN {X 0,Y 432.381,Z 417.625,A -85,B 0,C 180,E1 -9314.341,E2 -9314.341} C_VEL
LIN {X 0,Y 432.337,Z 417.63,A -85,B 0,C 180,E1 -9318.203,E2 -9318.203} C_VEL
LIN {X 0,Y 432.349,Z 417.632,A -85,B 0,C 180,E1 -9321.284,E2 -9321.284} C_VEL
LIN {X 0,Y 432.346,Z 417.631,A -85,B 0,C 180,E1 -9324.368,E2 -9324.368} C_VEL
LIN {X 0,Y 432.325,Z 417.632,A -85,B 0,C 180,E1 -9327.557,E2 -9327.557} C_VEL
LIN {X 0,Y 432.346,Z 417.633,A -85,B 0,C 180,E1 -9330.813,E2 -9330.813} C_VEL
LIN {X 0,Y 432.363,Z 417.627,A -85,B 0,C 180,E1 -9333.967,E2 -9333.967} C_VEL
LIN {X 0,Y 432.32,Z 417.635,A -85,B 0,C 180,E1 -9337.036,E2 -9337.036} C_VEL
LIN {X 0,Y 432.39,Z 417.627,A -85,B 0,C 180,E1 -9340.515,E2 -9340.515} C_VEL
LIN {X 0,Y 432.434,Z 417.618,A -85,B 0,C 180,E1 -9343.961,E2 -9343.961} C_VEL
LIN {X 0,Y 432.484,Z 417.612,A -85,B 0,C 180,E1 -9347.804,E2 -9347.804} C_VEL
LIN {X 0,Y 432.467,Z 417.614,A -85,B 0,C 180,E1 -9351.59,E2 -9351.59} C_VEL
LIN {X 0,Y 432.599,Z 417.601,A -85,B 0,C 180,E1 -9354.406,E2 -9354.406} C_VEL
LIN {X 0,Y 432.609,Z 417.6,A -85,B 0,C 180,E1 -9358.138,E2 -9358.138} C_VEL
LIN {X 0,Y 432.737,Z 417.582,A -85,B 0,C 180,E1 -9360,E2 -9360} C_VEL
LIN {X 0,Y 432.609,Z 417.599,A -85,B 0,C 180,E1 -9362.793,E2 -9362.793} C_VEL
LIN {X 0,Y 432.566,Z 417.605,A -85,B 0,C 180,E1 -9366.53,E2 -9366.53} C_VEL
LIN {X 0,Y 432.443,Z 417.617,A -85,B 0,C 180,E1 -9369.353,E2 -9369.353} C_VEL
LIN {X 0,Y 432.448,Z 417.617,A -85,B 0,C 180,E1 -9372.812,E2 -9372.812} C_VEL
LIN {X 0,Y 432.415,Z 417.624,A -85,B 0,C 180,E1 -9376.479,E2 -9376.479} C_VEL
LIN {X 0,Y 432.342,Z 417.633,A -85,B 0,C 180,E1 -9379.96,E2 -9379.96} C_VEL
LIN {X 0,Y 432.32,Z 417.632,A -85,B 0,C 180,E1 -9382.964,E2 -9382.964} C_VEL
LIN {X 0,Y 432.363,Z 417.631,A -85,B 0,C 180,E1 -9386.033,E2 -9386.033} C_VEL
LIN {X 0,Y 432.346,Z 417.629,A -85,B 0,C 180,E1 -9389.187,E2 -9389.187} C_VEL
LIN {X 0,Y 432.325,Z 417.634,A -85,B 0,C 180,E1 -9392.443,E2 -9392.443} C_VEL
LIN {X 0,Y 432.348,Z 417.632,A -85,B 0,C 180,E1 -9395.632,E2 -9395.632} C_VEL
LIN {X 0,Y 432.353,Z 417.628,A -85,B 0,C 180,E1 -9398.716,E2 -9398.716} C_VEL
LIN {X 0,Y 432.337,Z 417.634,A -85,B 0,C 180,E1 -9401.797,E2 -9401.797} C_VEL
LIN {X 0,Y 432.343,Z 417.634,A -85,B 0,C 180,E1 -9404.346,E2 -9404.346} C_VEL
LIN {X 0,Y 432.322,Z 417.635,A -85,B 0,C 180,E1 -9407.016,E2 -9407.016} C_VEL
LIN {X 0,Y 432.393,Z 417.789,A -85,B 0,C 180,E1 -9408.292,E2 -9408.292} C_VEL
LIN {X 0,Y 434.068,Z 426.313,A -85,B 0,C 180,E1 -9411.002,E2 -9411.002} C_VEL
LIN {X 0,Y 435.219,Z 432.413,A -85,B 0,C 180,E1 -9412.847,E2 -9412.847} C_VEL
LIN {X 0,Y 435.182,Z 437.022,A -85,B 0,C 180,E1 -9414.14,E2 -9414.14} C_VEL
LIN {X 0,Y 434.325,Z 450.395,A -85,B 0,C 180,E1 -9417.725,E2 -9417.725} C_VEL
LIN {X 0,Y 433.745,Z 461.659,A -85,B 0,C 180,E1 -9420.65,E2 -9420.65} C_VEL
LIN {X 0,Y 433.161,Z 474.902,A -85,B 0,C 180,E1 -9424.019,E2 -9424.019} C_VEL
LIN {X 0,Y 432.69,Z 486.983,A -85,B 0,C 180,E1 -9427.057,E2 -9427.057} C_VEL
LIN {X 0,Y 432.244,Z 500.969,A -85,B 0,C 180,E1 -9430.569,E2 -9430.569} C_VEL
LIN {X 0,Y 431.936,Z 511.812,A -85,B 0,C 180,E1 -9433.267,E2 -9433.267} C_VEL
LIN {X 0,Y 433.509,Z 526.292,A -85,B 0,C 180,E1 -9433.706,E2 -9433.706} C_VEL
LIN {X 0,Y 434.377,Z 539.196,A -85,B 0,C 180,E1 -9434.276,E2 -9434.276} C_VEL
LIN {X 0,Y 434.796,Z 546.902,A -85,B 0,C 180,E1 -9434.712,E2 -9434.712} C_VEL
LIN {X 0,Y 434.057,Z 558.313,A -85,B 0,C 180,E1 -9435.465,E2 -9435.465} C_VEL
LIN {X 0,Y 433.391,Z 569.932,A -85,B 0,C 180,E1 -9436.448,E2 -9436.448} C_VEL
LIN {X 0,Y 432.899,Z 580.537,A -85,B 0,C 180,E1 -9437.578,E2 -9437.578} C_VEL
LIN {X 0,Y 432.314,Z 589.545,A -85,B 0,C 180,E1 -9438.751,E2 -9438.751} C_VEL
LIN {X 0,Y 431.891,Z 598.375,A -85,B 0,C 180,E1 -9440.162,E2 -9440.162} C_VEL
LIN {X 0,Y 431.697,Z 605.464,A -85,B 0,C 180,E1 -9441.575,E2 -9441.575} C_VEL
LIN {X 0,Y 431.64,Z 611.169,A -85,B 0,C 180,E1 -9442.986,E2 -9442.986} C_VEL
LIN {X 0,Y 431.639,Z 615.653,A -85,B 0,C 180,E1 -9444.394,E2 -9444.394} C_VEL
LIN {X 0,Y 431.723,Z 618.039,A -85,B 0,C 180,E1 -9445.331,E2 -9445.331} C_VEL
LIN {X 0,Y 431.75,Z 619.97,A -85,B 0,C 180,E1 -9446.267,E2 -9446.267} C_VEL
LIN {X 0,Y 431.738,Z 621.414,A -85,B 0,C 180,E1 -9447.201,E2 -9447.201} C_VEL
LIN {X 0,Y 431.746,Z 622.446,A -85,B 0,C 180,E1 -9448.134,E2 -9448.134} C_VEL
LIN {X 0,Y 431.928,Z 623.325,A -85,B 0,C 180,E1 -9450,E2 -9450} C_VEL
LIN {X 0,Y 431.746,Z 622.447,A -85,B 0,C 180,E1 -9451.866,E2 -9451.866} C_VEL
LIN {X 0,Y 431.738,Z 621.415,A -85,B 0,C 180,E1 -9452.799,E2 -9452.799} C_VEL
LIN {X 0,Y 431.75,Z 619.971,A -85,B 0,C 180,E1 -9453.733,E2 -9453.733} C_VEL
LIN {X 0,Y 431.693,Z 616.925,A -85,B 0,C 180,E1 -9455.137,E2 -9455.137} C_VEL
LIN {X 0,Y 431.615,Z 612.448,A -85,B 0,C 180,E1 -9456.652,E2 -9456.652} C_VEL
LIN {X 0,Y 431.7,Z 606.5,A -85,B 0,C 180,E1 -9458.19,E2 -9458.19} C_VEL
LIN {X 0,Y 431.872,Z 599.635,A -85,B 0,C 180,E1 -9459.602,E2 -9459.602} C_VEL
LIN {X 0,Y 432.241,Z 591.156,A -85,B 0,C 180,E1 -9461.014,E2 -9461.014} C_VEL
LIN {X 0,Y 432.72,Z 582.492,A -85,B 0,C 180,E1 -9462.189,E2 -9462.189} C_VEL
LIN {X 0,Y 433.126,Z 573.492,A -85,B 0,C 180,E1 -9463.201,E2 -9463.201} C_VEL
LIN {X 0,Y 433.811,Z 562.737,A -85,B 0,C 180,E1 -9464.184,E2 -9464.184} C_VEL
LIN {X 0,Y 434.483,Z 551.58,A -85,B 0,C 180,E1 -9465,E2 -9465} C_VEL
LIN {X 0,Y 434.767,Z 543.772,A -85,B 0,C 180,E1 -9465.469,E2 -9465.469} C_VEL
LIN {X 0,Y 433.884,Z 531.408,A -85,B 0,C 180,E1 -9466.085,E2 -9466.085} C_VEL
LIN {X 0,Y 432.632,Z 517.709,A -85,B 0,C 180,E1 -9466.576,E2 -9466.576} C_VEL
LIN {X 0,Y 431.938,Z 511.489,A -85,B 0,C 180,E1 -9466.758,E2 -9466.758} C_VEL
LIN {X 0,Y 432.291,Z 498.838,A -85,B 0,C 180,E1 -9469.963,E2 -9469.963} C_VEL
LIN {X 0,Y 432.778,Z 484.965,A -85,B 0,C 180,E1 -9473.445,E2 -9473.445} C_VEL
LIN {X 0,Y 433.297,Z 471.395,A -85,B 0,C 180,E1 -9476.863,E2 -9476.863} C_VEL
LIN {X 0,Y 433.907,Z 458.563,A -85,B 0,C 180,E1 -9480.14,E2 -9480.14} C_VEL
LIN {X 0,Y 434.54,Z 446.269,A -85,B 0,C 180,E1 -9483.36,E2 -9483.36} C_VEL
LIN {X 0,Y 435.356,Z 434.032,A -85,B 0,C 180,E1 -9486.677,E2 -9486.677} C_VEL
LIN {X 0,Y 434.006,Z 425.722,A -85,B 0,C 180,E1 -9489.164,E2 -9489.164} C_VEL
LIN {X 0,Y 432.378,Z 417.625,A -85,B 0,C 180,E1 -9491.792,E2 -9491.792} C_VEL
LIN {X 0,Y 432.336,Z 417.633,A -85,B 0,C 180,E1 -9494.347,E2 -9494.347} C_VEL
LIN {X 0,Y 432.328,Z 417.635,A -85,B 0,C 180,E1 -9497.015,E2 -9497.015} C_VEL
LIN {X 0,Y 432.34,Z 417.632,A -85,B 0,C 180,E1 -9499.82,E2 -9499.82} C_VEL
LIN {X 0,Y 432.319,Z 417.632,A -85,B 0,C 180,E1 -9503.023,E2 -9503.023} C_VEL
LIN {X 0,Y 432.363,Z 417.631,A -85,B 0,C 180,E1 -9505.997,E2 -9505.997} C_VEL
LIN {X 0,Y 432.351,Z 417.63,A -85,B 0,C 180,E1 -9509.49,E2 -9509.49} C_VEL
LIN {X 0,Y 432.395,Z 417.622,A -85,B 0,C 180,E1 -9512.928,E2 -9512.928} C_VEL
LIN {X 0,Y 432.371,Z 417.63,A -85,B 0,C 180,E1 -9516.023,E2 -9516.023} C_VEL
LIN {X 0,Y 432.354,Z 417.628,A -85,B 0,C 180,E1 -9519.046,E2 -9519.046} C_VEL
LIN {X 0,Y 432.383,Z 417.628,A -85,B 0,C 180,E1 -9522.011,E2 -9522.011} C_VEL
LIN {X 0,Y 432.399,Z 417.622,A -85,B 0,C 180,E1 -9524.927,E2 -9524.927} C_VEL
LIN {X 0,Y 432.484,Z 417.616,A -85,B 0,C 180,E1 -9527.804,E2 -9527.804} C_VEL
LIN {X 0,Y 432.467,Z 417.618,A -85,B 0,C 180,E1 -9531.59,E2 -9531.59} C_VEL
LIN {X 0,Y 432.601,Z 417.598,A -85,B 0,C 180,E1 -9534.406,E2 -9534.406} C_VEL
LIN {X 0,Y 432.611,Z 417.597,A -85,B 0,C 180,E1 -9538.138,E2 -9538.138} C_VEL
LIN {X 0,Y 432.738,Z 417.582,A -85,B 0,C 180,E1 -9540,E2 -9540} C_VEL
LIN {X 0,Y 432.597,Z 417.598,A -85,B 0,C 180,E1 -9542.794,E2 -9542.794} C_VEL
LIN {X 0,Y 432.565,Z 417.602,A -85,B 0,C 180,E1 -9546.531,E2 -9546.531} C_VEL
LIN {X 0,Y 432.446,Z 417.62,A -85,B 0,C 180,E1 -9549.353,E2 -9549.353} C_VEL
LIN {X 0,Y 432.449,Z 417.617,A -85,B 0,C 180,E1 -9552.812,E2 -9552.812} C_VEL
LIN {X 0,Y 432.417,Z 417.62,A -85,B 0,C 180,E1 -9556.479,E2 -9556.479} C_VEL
LIN {X 0,Y 432.343,Z 417.631,A -85,B 0,C 180,E1 -9559.96,E2 -9559.96} C_VEL
LIN {X 0,Y 432.323,Z 417.635,A -85,B 0,C 180,E1 -9562.964,E2 -9562.964} C_VEL
LIN {X 0,Y 432.368,Z 417.627,A -85,B 0,C 180,E1 -9566.032,E2 -9566.032} C_VEL
LIN {X 0,Y 432.347,Z 417.633,A -85,B 0,C 180,E1 -9569.187,E2 -9569.187} C_VEL
LIN {X 0,Y 432.327,Z 417.631,A -85,B 0,C 180,E1 -9572.443,E2 -9572.443} C_VEL
LIN {X 0,Y 432.347,Z 417.631,A -85,B 0,C 180,E1 -9575.632,E2 -9575.632} C_VEL
LIN {X 0,Y 432.344,Z 417.632,A -85,B 0,C 180,E1 -9578.714,E2 -9578.714} C_VEL
LIN {X 0,Y 432.338,Z 417.63,A -85,B 0,C 180,E1 -9581.797,E2 -9581.797} C_VEL
LIN {X 0,Y 432.382,Z 417.625,A -85,B 0,C 180,E1 -9585.659,E2 -9585.659} C_VEL
LIN {X 0,Y 432.377,Z 417.626,A -85,B 0,C 180,E1 -9588.392,E2 -9588.392} C_VEL
LIN {X 0,Y 432.356,Z 417.628,A -85,B 0,C 180,E1 -9591.852,E2 -9591.852} C_VEL
LIN {X 0,Y 432.343,Z 417.631,A -85,B 0,C 180,E1 -9595.323,E2 -9595.323} C_VEL
LIN {X 0,Y 432.325,Z 417.636,A -85,B 0,C 180,E1 -9598.654,E2 -9598.654} C_VEL
LIN {X 0,Y 432.386,Z 417.624,A -85,B 0,C 180,E1 -9601.877,E2 -9601.877} C_VEL
LIN {X 0,Y 432.355,Z 417.631,A -85,B 0,C 180,E1 -9604.999,E2 -9604.999} C_VEL
LIN {X 0,Y 432.362,Z 417.628,A -85,B 0,C 180,E1 -9608.046,E2 -9608.046} C_VEL
LIN {X 0,Y 432.39,Z 417.626,A -85,B 0,C 180,E1 -9611.03,E2 -9611.03} C_VEL
LIN {X 0,Y 432.423,Z 417.64,A -85,B 0,C 180,E1 -9614.142,E2 -9614.142} C_VEL
LIN {X 0,Y 435.748,Z 428.917,A -85,B 0,C 180,E1 -9614.925,E2 -9614.925} C_VEL
LIN {X 0,Y 436.358,Z 432.109,A -85,B 0,C 180,E1 -9615.171,E2 -9615.171} C_VEL
LIN {X 0,Y 435.802,Z 442.996,A -85,B 0,C 180,E1 -9616.001,E2 -9616.001} C_VEL
LIN {X 0,Y 435.206,Z 453.848,A -85,B 0,C 180,E1 -9617.052,E2 -9617.052} C_VEL
LIN {X 0,Y 434.588,Z 464.371,A -85,B 0,C 180,E1 -9618.337,E2 -9618.337} C_VEL
LIN {X 0,Y 434.074,Z 472.122,A -85,B 0,C 180,E1 -9619.505,E2 -9619.505} C_VEL
LIN {X 0,Y 433.485,Z 479.699,A -85,B 0,C 180,E1 -9620.905,E2 -9620.905} C_VEL
LIN {X 0,Y 433.175,Z 484.976,A -85,B 0,C 180,E1 -9622.107,E2 -9622.107} C_VEL
LIN {X 0,Y 432.908,Z 489.825,A -85,B 0,C 180,E1 -9623.475,E2 -9623.475} C_VEL
LIN {X 0,Y 432.524,Z 493.714,A -85,B 0,C 180,E1 -9624.873,E2 -9624.873} C_VEL
LIN {X 0,Y 432.28,Z 496.58,A -85,B 0,C 180,E1 -9626.271,E2 -9626.271} C_VEL
LIN {X 0,Y 432.14,Z 497.958,A -85,B 0,C 180,E1 -9627.203,E2 -9627.203} C_VEL
LIN {X 0,Y 432.164,Z 498.918,A -85,B 0,C 180,E1 -9628.136,E2 -9628.136} C_VEL
LIN {X 0,Y 432.084,Z 499.594,A -85,B 0,C 180,E1 -9629.362,E2 -9629.362} C_VEL
LIN {X 0,Y 431.443,Z 499.837,A -85,B 0,C 180,E1 -9630.141,E2 -9630.141} C_VEL
LIN {X 0,Y 428.583,Z 499.842,A -85,B 0,C 180,E1 -9631.407,E2 -9631.407} C_VEL
LIN {X 0,Y 425.763,Z 499.169,A -85,B 0,C 180,E1 -9632.684,E2 -9632.684} C_VEL
LIN {X 0,Y 425.197,Z 498.191,A -85,B 0,C 180,E1 -9633.469,E2 -9633.469} C_VEL
LIN {X 0,Y 425.519,Z 494.93,A -85,B 0,C 180,E1 -9635.212,E2 -9635.212} C_VEL
LIN {X 0,Y 425.911,Z 491.113,A -85,B 0,C 180,E1 -9636.633,E2 -9636.633} C_VEL
LIN {X 0,Y 426.152,Z 485.238,A -85,B 0,C 180,E1 -9638.306,E2 -9638.306} C_VEL
LIN {X 0,Y 426.731,Z 478.821,A -85,B 0,C 180,E1 -9639.719,E2 -9639.719} C_VEL
LIN {X 0,Y 427.363,Z 470.799,A -85,B 0,C 180,E1 -9641.141,E2 -9641.141} C_VEL
LIN {X 0,Y 427.894,Z 462.581,A -85,B 0,C 180,E1 -9642.329,E2 -9642.329} C_VEL
LIN {X 0,Y 428.537,Z 452.399,A -85,B 0,C 180,E1 -9643.515,E2 -9643.515} C_VEL
LIN {X 0,Y 429.153,Z 441.906,A -85,B 0,C 180,E1 -9644.496,E2 -9644.496} C_VEL
LIN {X 0,Y 429.515,Z 432.974,A -85,B 0,C 180,E1 -9645.177,E2 -9645.177} C_VEL
LIN {X 0,Y 426.299,Z 421.637,A -85,B 0,C 180,E1 -9646.03,E2 -9646.03} C_VEL
LIN {X 0,Y 425.399,Z 418.496,A -85,B 0,C 180,E1 -9646.25,E2 -9646.25} C_VEL
LIN {X 0,Y 425.331,Z 418.506,A -85,B 0,C 180,E1 -9649.635,E2 -9649.635} C_VEL
LIN {X 0,Y 425.311,Z 418.509,A -85,B 0,C 180,E1 -9653.365,E2 -9653.365} C_VEL
LIN {X 0,Y 425.352,Z 418.503,A -85,B 0,C 180,E1 -9656.845,E2 -9656.845} C_VEL
LIN {X 0,Y 425.294,Z 418.508,A -85,B 0,C 180,E1 -9659.719,E2 -9659.719} C_VEL
LIN {X 0,Y 425.285,Z 418.513,A -85,B 0,C 180,E1 -9663.048,E2 -9663.048} C_VEL
LIN {X 0,Y 425.288,Z 418.508,A -85,B 0,C 180,E1 -9665.929,E2 -9665.929} C_VEL
LIN {X 0,Y 425.317,Z 418.509,A -85,B 0,C 180,E1 -9669.046,E2 -9669.046} C_VEL
LIN {X 0,Y 425.334,Z 418.505,A -85,B 0,C 180,E1 -9672.646,E2 -9672.646} C_VEL
LIN {X 0,Y 425.271,Z 418.509,A -85,B 0,C 180,E1 -9676.045,E2 -9676.045} C_VEL
LIN {X 0,Y 425.278,Z 418.512,A -85,B 0,C 180,E1 -9678.622,E2 -9678.622} C_VEL
LIN {X 0,Y 425.312,Z 418.509,A -85,B 0,C 180,E1 -9681.103,E2 -9681.103} C_VEL
LIN {X 0,Y 425.302,Z 418.51,A -85,B 0,C 180,E1 -9684.664,E2 -9684.664} C_VEL
LIN {X 0,Y 425.267,Z 418.511,A -85,B 0,C 180,E1 -9688.073,E2 -9688.073} C_VEL
LIN {X 0,Y 425.334,Z 418.503,A -85,B 0,C 180,E1 -9691.368,E2 -9691.368} C_VEL
LIN {X 0,Y 425.356,Z 418.5,A -85,B 0,C 180,E1 -9693.505,E2 -9693.505} C_VEL
LIN {X 0,Y 425.307,Z 418.51,A -85,B 0,C 180,E1 -9696.635,E2 -9696.635} C_VEL
LIN {X 0,Y 425.332,Z 418.506,A -85,B 0,C 180,E1 -9700.364,E2 -9700.364} C_VEL
LIN {X 0,Y 425.391,Z 418.494,A -85,B 0,C 180,E1 -9703.688,E2 -9703.688} C_VEL
LIN {X 0,Y 425.433,Z 418.49,A -85,B 0,C 180,E1 -9707.599,E2 -9707.599} C_VEL
LIN {X 0,Y 425.411,Z 418.493,A -85,B 0,C 180,E1 -9711.449,E2 -9711.449} C_VEL
LIN {X 0,Y 425.555,Z 418.478,A -85,B 0,C 180,E1 -9714.313,E2 -9714.313} C_VEL
LIN {X 0,Y 425.579,Z 418.475,A -85,B 0,C 180,E1 -9718.107,E2 -9718.107} C_VEL
LIN {X 0,Y 425.707,Z 418.458,A -85,B 0,C 180,E1 -9720,E2 -9720} C_VEL
LIN {X 0,Y 425.561,Z 418.476,A -85,B 0,C 180,E1 -9722.84,E2 -9722.84} C_VEL
LIN {X 0,Y 425.522,Z 418.482,A -85,B 0,C 180,E1 -9726.639,E2 -9726.639} C_VEL
LIN {X 0,Y 425.403,Z 418.494,A -85,B 0,C 180,E1 -9729.509,E2 -9729.509} C_VEL
LIN {X 0,Y 425.407,Z 418.493,A -85,B 0,C 180,E1 -9732.91,E2 -9732.91} C_VEL
LIN {X 0,Y 425.364,Z 418.501,A -85,B 0,C 180,E1 -9736.605,E2 -9736.605} C_VEL
LIN {X 0,Y 425.331,Z 418.504,A -85,B 0,C 180,E1 -9739.636,E2 -9739.636} C_VEL
LIN {X 0,Y 425.29,Z 418.511,A -85,B 0,C 180,E1 -9742.339,E2 -9742.339} C_VEL
LIN {X 0,Y 425.293,Z 418.508,A -85,B 0,C 180,E1 -9745.446,E2 -9745.446} C_VEL
LIN {X 0,Y 425.351,Z 418.501,A -85,B 0,C 180,E1 -9747.558,E2 -9747.558} C_VEL
LIN {X 0,Y 425.29,Z 418.508,A -85,B 0,C 180,E1 -9750.816,E2 -9750.816} C_VEL
LIN {X 0,Y 425.314,Z 418.508,A -85,B 0,C 180,E1 -9754.288,E2 -9754.288} C_VEL
LIN {X 0,Y 425.288,Z 418.512,A -85,B 0,C 180,E1 -9757.693,E2 -9757.693} C_VEL
LIN {X 0,Y 425.284,Z 418.509,A -85,B 0,C 180,E1 -9760.521,E2 -9760.521} C_VEL
LIN {X 0,Y 425.266,Z 418.515,A -85,B 0,C 180,E1 -9763.352,E2 -9763.352} C_VEL
LIN {X 0,Y 425.26,Z 418.517,A -85,B 0,C 180,E1 -9766.649,E2 -9766.649} C_VEL
LIN {X 0,Y 425.337,Z 418.69,A -85,B 0,C 180,E1 -9767.974,E2 -9767.974} C_VEL
LIN {X 0,Y 427.028,Z 426.981,A -85,B 0,C 180,E1 -9770.672,E2 -9770.672} C_VEL
LIN {X 0,Y 428.401,Z 434.997,A -85,B 0,C 180,E1 -9773.124,E2 -9773.124} C_VEL
LIN {X 0,Y 427.687,Z 445.489,A -85,B 0,C 180,E1 -9776.033,E2 -9776.033} C_VEL
LIN {X 0,Y 427.033,Z 457.74,A -85,B 0,C 180,E1 -9779.323,E2 -9779.323} C_VEL
LIN {X 0,Y 426.31,Z 471.446,A -85,B 0,C 180,E1 -9782.902,E2 -9782.902} C_VEL
LIN {X 0,Y 425.765,Z 484.048,A -85,B 0,C 180,E1 -9786.145,E2 -9786.145} C_VEL
LIN {X 0,Y 425.242,Z 497.884,A -85,B 0,C 180,E1 -9789.692,E2 -9789.692} C_VEL
LIN {X 0,Y 424.872,Z 509.434,A -85,B 0,C 180,E1 -9792.678,E2 -9792.678} C_VEL
LIN {X 0,Y 424.855,Z 510.501,A -85,B 0,C 180,E1 -9792.956,E2 -9792.956} C_VEL
LIN {X 0,Y 426.579,Z 526.221,A -85,B 0,C 180,E1 -9793.466,E2 -9793.466} C_VEL
LIN {X 0,Y 427.399,Z 539.312,A -85,B 0,C 180,E1 -9794.074,E2 -9794.074} C_VEL
LIN {X 0,Y 427.84,Z 546.885,A -85,B 0,C 180,E1 -9794.518,E2 -9794.518} C_VEL
LIN {X 0,Y 427.035,Z 558.854,A -85,B 0,C 180,E1 -9795.343,E2 -9795.343} C_VEL
LIN {X 0,Y 426.323,Z 570.821,A -85,B 0,C 180,E1 -9796.414,E2 -9796.414} C_VEL
LIN {X 0,Y 425.759,Z 581.495,A -85,B 0,C 180,E1 -9797.608,E2 -9797.608} C_VEL
LIN {X 0,Y 425.195,Z 590.145,A -85,B 0,C 180,E1 -9798.801,E2 -9798.801} C_VEL
LIN {X 0,Y 424.806,Z 598.622,A -85,B 0,C 180,E1 -9800.237,E2 -9800.237} C_VEL
LIN {X 0,Y 424.618,Z 605.486,A -85,B 0,C 180,E1 -9801.673,E2 -9801.673} C_VEL
LIN {X 0,Y 424.541,Z 611.794,A -85,B 0,C 180,E1 -9803.346,E2 -9803.346} C_VEL
LIN {X 0,Y 424.629,Z 615.914,A -85,B 0,C 180,E1 -9804.777,E2 -9804.777} C_VEL
LIN {X 0,Y 424.711,Z 618.961,A -85,B 0,C 180,E1 -9806.205,E2 -9806.205} C_VEL
LIN {X 0,Y 424.695,Z 620.406,A -85,B 0,C 180,E1 -9807.154,E2 -9807.154} C_VEL
LIN {X 0,Y 424.709,Z 621.439,A -85,B 0,C 180,E1 -9808.103,E2 -9808.103} C_VEL
LIN {X 0,Y 424.906,Z 622.321,A -85,B 0,C 180,E1 -9810,E2 -9810} C_VEL
LIN {X 0,Y 424.709,Z 621.44,A -85,B 0,C 180,E1 -9811.897,E2 -9811.897} C_VEL
LIN {X 0,Y 424.695,Z 620.406,A -85,B 0,C 180,E1 -9812.846,E2 -9812.846} C_VEL
LIN {X 0,Y 424.711,Z 618.961,A -85,B 0,C 180,E1 -9813.795,E2 -9813.795} C_VEL
LIN {X 0,Y 424.629,Z 615.91,A -85,B 0,C 180,E1 -9815.223,E2 -9815.223} C_VEL
LIN {X 0,Y 424.541,Z 611.785,A -85,B 0,C 180,E1 -9816.655,E2 -9816.655} C_VEL
LIN {X 0,Y 424.618,Z 605.475,A -85,B 0,C 180,E1 -9818.327,E2 -9818.327} C_VEL
LIN {X 0,Y 424.806,Z 598.608,A -85,B 0,C 180,E1 -9819.763,E2 -9819.763} C_VEL
LIN {X 0,Y 425.196,Z 590.127,A -85,B 0,C 180,E1 -9821.199,E2 -9821.199} C_VEL
LIN {X 0,Y 425.757,Z 581.471,A -85,B 0,C 180,E1 -9822.392,E2 -9822.392} C_VEL
LIN {X 0,Y 426.327,Z 570.79,A -85,B 0,C 180,E1 -9823.587,E2 -9823.587} C_VEL
LIN {X 0,Y 427.031,Z 558.816,A -85,B 0,C 180,E1 -9824.658,E2 -9824.658} C_VEL
LIN {X 0,Y 427.844,Z 546.824,A -85,B 0,C 180,E1 -9825.482,E2 -9825.482} C_VEL
LIN {X 0,Y 427.085,Z 534.159,A -85,B 0,C 180,E1 -9826.184,E2 -9826.184} C_VEL
LIN {X 0,Y 426.121,Z 521.6,A -85,B 0,C 180,E1 -9826.7,E2 -9826.7} C_VEL
LIN {X 0,Y 424.866,Z 510.468,A -85,B 0,C 180,E1 -9827.044,E2 -9827.044} C_VEL
LIN {X 0,Y 425.198,Z 499.491,A -85,B 0,C 180,E1 -9829.886,E2 -9829.886} C_VEL
LIN {X 0,Y 425.7,Z 486.011,A -85,B 0,C 180,E1 -9833.342,E2 -9833.342} C_VEL
LIN {X 0,Y 426.224,Z 472.695,A -85,B 0,C 180,E1 -9836.766,E2 -9836.766} C_VEL
LIN {X 0,Y 426.871,Z 459.739,A -85,B 0,C 180,E1 -9840.143,E2 -9840.143} C_VEL
LIN {X 0,Y 427.519,Z 448.9,A -85,B 0,C 180,E1 -9843.029,E2 -9843.029} C_VEL
LIN {X 0,Y 428.367,Z 436.297,A -85,B 0,C 180,E1 -9846.494,E2 -9846.494} C_VEL
LIN {X 0,Y 427.849,Z 431.359,A -85,B 0,C 180,E1 -9847.958,E2 -9847.958} C_VEL
LIN {X 0,Y 426.199,Z 422.761,A -85,B 0,C 180,E1 -9850.664,E2 -9850.664} C_VEL
LIN {X 0,Y 425.32,Z 418.504,A -85,B 0,C 180,E1 -9852.123,E2 -9852.123} C_VEL
LIN {X 0,Y 425.292,Z 418.509,A -85,B 0,C 180,E1 -9855.282,E2 -9855.282} C_VEL
LIN {X 0,Y 425.279,Z 418.514,A -85,B 0,C 180,E1 -9858.622,E2 -9858.622} C_VEL
LIN {X 0,Y 425.316,Z 418.504,A -85,B 0,C 180,E1 -9861.103,E2 -9861.103} C_VEL
LIN {X 0,Y 425.304,Z 418.507,A -85,B 0,C 180,E1 -9864.664,E2 -9864.664} C_VEL
LIN {X 0,Y 425.269,Z 418.515,A -85,B 0,C 180,E1 -9868.073,E2 -9868.073} C_VEL
LIN {X 0,Y 425.335,Z 418.503,A -85,B 0,C 180,E1 -9871.368,E2 -9871.368} C_VEL
LIN {X 0,Y 425.357,Z 418.501,A -85,B 0,C 180,E1 -9873.506,E2 -9873.506} C_VEL
LIN {X 0,Y 425.288,Z 418.508,A -85,B 0,C 180,E1 -9876.634,E2 -9876.634} C_VEL
LIN {X 0,Y 425.299,Z 418.51,A -85,B 0,C 180,E1 -9879.695,E2 -9879.695} C_VEL
LIN {X 0,Y 425.346,Z 418.501,A -85,B 0,C 180,E1 -9882.698,E2 -9882.698} C_VEL
LIN {X 0,Y 425.358,Z 418.503,A -85,B 0,C 180,E1 -9885.65,E2 -9885.65} C_VEL
LIN {X 0,Y 425.37,Z 418.498,A -85,B 0,C 180,E1 -9888.564,E2 -9888.564} C_VEL
LIN {X 0,Y 425.509,Z 418.482,A -85,B 0,C 180,E1 -9892.311,E2 -9892.311} C_VEL
LIN {X 0,Y 425.556,Z 418.476,A -85,B 0,C 180,E1 -9894.313,E2 -9894.313} C_VEL
LIN {X 0,Y 425.58,Z 418.473,A -85,B 0,C 180,E1 -9898.107,E2 -9898.107} C_VEL
LIN {X 0,Y 425.708,Z 418.458,A -85,B 0,C 180,E1 -9900,E2 -9900} C_VEL
LIN {X 0,Y 425.55,Z 418.475,A -85,B 0,C 180,E1 -9902.84,E2 -9902.84} C_VEL
LIN {X 0,Y 425.554,Z 418.479,A -85,B 0,C 180,E1 -9905.687,E2 -9905.687} C_VEL
LIN {X 0,Y 425.412,Z 418.492,A -85,B 0,C 180,E1 -9908.551,E2 -9908.551} C_VEL
LIN {X 0,Y 425.434,Z 418.489,A -85,B 0,C 180,E1 -9912.401,E2 -9912.401} C_VEL
LIN {X 0,Y 425.392,Z 418.494,A -85,B 0,C 180,E1 -9916.312,E2 -9916.312} C_VEL
LIN {X 0,Y 425.333,Z 418.506,A -85,B 0,C 180,E1 -9919.636,E2 -9919.636} C_VEL
LIN {X 0,Y 425.31,Z 418.51,A -85,B 0,C 180,E1 -9923.365,E2 -9923.365} C_VEL
LIN {X 0,Y 425.352,Z 418.502,A -85,B 0,C 180,E1 -9926.844,E2 -9926.844} C_VEL
LIN {X 0,Y 425.295,Z 418.509,A -85,B 0,C 180,E1 -9929.719,E2 -9929.719} C_VEL
LIN {X 0,Y 425.286,Z 418.512,A -85,B 0,C 180,E1 -9933.048,E2 -9933.048} C_VEL
LIN {X 0,Y 425.285,Z 418.509,A -85,B 0,C 180,E1 -9935.929,E2 -9935.929} C_VEL
LIN {X 0,Y 425.291,Z 418.512,A -85,B 0,C 180,E1 -9939.042,E2 -9939.042} C_VEL
LIN {X 0,Y 425.295,Z 418.507,A -85,B 0,C 180,E1 -9941.958,E2 -9941.958} C_VEL
LIN {X 0,Y 425.318,Z 418.508,A -85,B 0,C 180,E1 -9945.279,E2 -9945.279} C_VEL
LIN {X 0,Y 425.314,Z 418.507,A -85,B 0,C 180,E1 -9948.626,E2 -9948.626} C_VEL
LIN {X 0,Y 425.328,Z 418.507,A -85,B 0,C 180,E1 -9951.104,E2 -9951.104} C_VEL
LIN {X 0,Y 425.303,Z 418.51,A -85,B 0,C 180,E1 -9954.664,E2 -9954.664} C_VEL
LIN {X 0,Y 425.268,Z 418.51,A -85,B 0,C 180,E1 -9958.073,E2 -9958.073} C_VEL
LIN {X 0,Y 425.335,Z 418.504,A -85,B 0,C 180,E1 -9961.368,E2 -9961.368} C_VEL
LIN {X 0,Y 425.299,Z 418.51,A -85,B 0,C 180,E1 -9964.555,E2 -9964.555} C_VEL
LIN {X 0,Y 425.291,Z 418.508,A -85,B 0,C 180,E1 -9967.661,E2 -9967.661} C_VEL
LIN {X 0,Y 425.365,Z 418.502,A -85,B 0,C 180,E1 -9970.704,E2 -9970.704} C_VEL
LIN {X 0,Y 425.433,Z 418.69,A -85,B 0,C 180,E1 -9973.875,E2 -9973.875} C_VEL
LIN {X 0,Y 428.794,Z 429.955,A -85,B 0,C 180,E1 -9974.675,E2 -9974.675} C_VEL
LIN {X 0,Y 429.558,Z 433.224,A -85,B 0,C 180,E1 -9974.938,E2 -9974.938} C_VEL
LIN {X 0,Y 428.988,Z 444.006,A -85,B 0,C 180,E1 -9975.774,E2 -9975.774} C_VEL
LIN {X 0,Y 428.361,Z 454.857,A -85,B 0,C 180,E1 -9976.841,E2 -9976.841} C_VEL
LIN {X 0,Y 427.709,Z 465.379,A -85,B 0,C 180,E1 -9978.147,E2 -9978.147} C_VEL
LIN {X 0,Y 427.168,Z 473.129,A -85,B 0,C 180,E1 -9979.333,E2 -9979.333} C_VEL
LIN {X 0,Y 426.547,Z 480.707,A -85,B 0,C 180,E1 -9980.755,E2 -9980.755} C_VEL
LIN {X 0,Y 426.215,Z 485.981,A -85,B 0,C 180,E1 -9981.977,E2 -9981.977} C_VEL
LIN {X 0,Y 425.932,Z 490.83,A -85,B 0,C 180,E1 -9983.367,E2 -9983.367} C_VEL
LIN {X 0,Y 425.526,Z 494.72,A -85,B 0,C 180,E1 -9984.788,E2 -9984.788} C_VEL
LIN {X 0,Y 425.267,Z 497.586,A -85,B 0,C 180,E1 -9986.21,E2 -9986.21} C_VEL
LIN {X 0,Y 425.121,Z 498.963,A -85,B 0,C 180,E1 -9987.157,E2 -9987.157} C_VEL
LIN {X 0,Y 425.143,Z 499.923,A -85,B 0,C 180,E1 -9988.105,E2 -9988.105} C_VEL
LIN {X 0,Y 425.133,Z 500.746,A -85,B 0,C 180,E1 -9990,E2 -9990} C_VEL
LIN {X 0,Y 425.051,Z 500.576,A -85,B 0,C 180,E1 -9990.947,E2 -9990.947} C_VEL
LIN {X 0,Y 425.142,Z 499.999,A -85,B 0,C 180,E1 -9991.895,E2 -9991.895} C_VEL
LIN {X 0,Y 425.197,Z 498.191,A -85,B 0,C 180,E1 -9993.469,E2 -9993.469} C_VEL
LIN {X 0,Y 424.693,Z 497.047,A -85,B 0,C 180,E1 -9994.246,E2 -9994.246} C_VEL
LIN {X 0,Y 422.153,Z 494.842,A -85,B 0,C 180,E1 -9995.507,E2 -9995.507} C_VEL
LIN {X 0,Y 419.982,Z 492.596,A -85,B 0,C 180,E1 -9996.504,E2 -9996.504} C_VEL
LIN {X 0,Y 419.086,Z 490.503,A -85,B 0,C 180,E1 -9997.251,E2 -9997.251} C_VEL
LIN {X 0,Y 419.035,Z 489.689,A -85,B 0,C 180,E1 -9997.499,E2 -9997.499} C_VEL
LIN {X 0,Y 419.381,Z 484.31,A -85,B 0,C 180,E1 -9998.917,E2 -9998.917} C_VEL
LIN {X 0,Y 419.991,Z 477.356,A -85,B 0,C 180,E1 -10000.363,E2 -10000.363} C_VEL
LIN {X 0,Y 420.675,Z 468.687,A -85,B 0,C 180,E1 -10001.809,E2 -10001.809} C_VEL
LIN {X 0,Y 421.256,Z 459.785,A -85,B 0,C 180,E1 -10003.016,E2 -10003.016} C_VEL
LIN {X 0,Y 421.916,Z 449.891,A -85,B 0,C 180,E1 -10004.1,E2 -10004.1} C_VEL
LIN {X 0,Y 422.504,Z 438.75,A -85,B 0,C 180,E1 -10005.075,E2 -10005.075} C_VEL
LIN {X 0,Y 422.613,Z 433.99,A -85,B 0,C 180,E1 -10005.431,E2 -10005.431} C_VEL
LIN {X 0,Y 419.312,Z 422.669,A -85,B 0,C 180,E1 -10006.305,E2 -10006.305} C_VEL
LIN {X 0,Y 418.341,Z 419.375,A -85,B 0,C 180,E1 -10006.532,E2 -10006.532} C_VEL
LIN {X 0,Y 418.273,Z 419.386,A -85,B 0,C 180,E1 -10009.79,E2 -10009.79} C_VEL
LIN {X 0,Y 418.241,Z 419.387,A -85,B 0,C 180,E1 -10012.736,E2 -10012.736} C_VEL
LIN {X 0,Y 418.274,Z 419.382,A -85,B 0,C 180,E1 -10015.904,E2 -10015.904} C_VEL
LIN {X 0,Y 418.267,Z 419.386,A -85,B 0,C 180,E1 -10019.162,E2 -10019.162} C_VEL
LIN {X 0,Y 418.26,Z 419.386,A -85,B 0,C 180,E1 -10022.844,E2 -10022.844} C_VEL
LIN {X 0,Y 418.252,Z 419.384,A -85,B 0,C 180,E1 -10026.239,E2 -10026.239} C_VEL
LIN {X 0,Y 418.269,Z 419.383,A -85,B 0,C 180,E1 -10029.68,E2 -10029.68} C_VEL
LIN {X 0,Y 418.288,Z 419.38,A -85,B 0,C 180,E1 -10032.33,E2 -10032.33} C_VEL
LIN {X 0,Y 418.258,Z 419.388,A -85,B 0,C 180,E1 -10035.111,E2 -10035.111} C_VEL
LIN {X 0,Y 418.245,Z 419.385,A -85,B 0,C 180,E1 -10037.767,E2 -10037.767} C_VEL
LIN {X 0,Y 418.258,Z 419.386,A -85,B 0,C 180,E1 -10040.619,E2 -10040.619} C_VEL
LIN {X 0,Y 418.245,Z 419.385,A -85,B 0,C 180,E1 -10043.976,E2 -10043.976} C_VEL
LIN {X 0,Y 418.26,Z 419.386,A -85,B 0,C 180,E1 -10047.156,E2 -10047.156} C_VEL
LIN {X 0,Y 418.271,Z 419.386,A -85,B 0,C 180,E1 -10050.895,E2 -10050.895} C_VEL
LIN {X 0,Y 418.271,Z 419.382,A -85,B 0,C 180,E1 -10054.096,E2 -10054.096} C_VEL
LIN {X 0,Y 418.24,Z 419.387,A -85,B 0,C 180,E1 -10057.264,E2 -10057.264} C_VEL
LIN {X 0,Y 418.286,Z 419.383,A -85,B 0,C 180,E1 -10060.364,E2 -10060.364} C_VEL
LIN {X 0,Y 418.32,Z 419.375,A -85,B 0,C 180,E1 -10063.405,E2 -10063.405} C_VEL
LIN {X 0,Y 418.358,Z 419.373,A -85,B 0,C 180,E1 -10066.994,E2 -10066.994} C_VEL
LIN {X 0,Y 418.345,Z 419.376,A -85,B 0,C 180,E1 -10070.329,E2 -10070.329} C_VEL
LIN {X 0,Y 418.482,Z 419.356,A -85,B 0,C 180,E1 -10073.249,E2 -10073.249} C_VEL
LIN {X 0,Y 418.342,Z 419.373,A -85,B 0,C 180,E1 -10075.182,E2 -10075.182} C_VEL
LIN {X 0,Y 418.548,Z 419.35,A -85,B 0,C 180,E1 -10078.075,E2 -10078.075} C_VEL
LIN {X 0,Y 418.676,Z 419.333,A -85,B 0,C 180,E1 -10080,E2 -10080} C_VEL
LIN {X 0,Y 418.514,Z 419.353,A -85,B 0,C 180,E1 -10082.888,E2 -10082.888} C_VEL
LIN {X 0,Y 418.513,Z 419.353,A -85,B 0,C 180,E1 -10085.783,E2 -10085.783} C_VEL
LIN {X 0,Y 418.38,Z 419.371,A -85,B 0,C 180,E1 -10088.695,E2 -10088.695} C_VEL
LIN {X 0,Y 418.333,Z 419.375,A -85,B 0,C 180,E1 -10091.631,E2 -10091.631} C_VEL
LIN {X 0,Y 418.309,Z 419.379,A -85,B 0,C 180,E1 -10094.597,E2 -10094.597} C_VEL
LIN {X 0,Y 418.291,Z 419.38,A -85,B 0,C 180,E1 -10097.604,E2 -10097.604} C_VEL
LIN {X 0,Y 418.253,Z 419.386,A -85,B 0,C 180,E1 -10100.663,E2 -10100.663} C_VEL
LIN {X 0,Y 418.277,Z 419.385,A -85,B 0,C 180,E1 -10103.782,E2 -10103.782} C_VEL
LIN {X 0,Y 418.312,Z 419.376,A -85,B 0,C 180,E1 -10107.07,E2 -10107.07} C_VEL
LIN {X 0,Y 418.247,Z 419.389,A -85,B 0,C 180,E1 -10110.272,E2 -10110.272} C_VEL
LIN {X 0,Y 418.251,Z 419.387,A -85,B 0,C 180,E1 -10113.677,E2 -10113.677} C_VEL
LIN {X 0,Y 418.248,Z 419.385,A -85,B 0,C 180,E1 -10117.223,E2 -10117.223} C_VEL
LIN {X 0,Y 418.254,Z 419.388,A -85,B 0,C 180,E1 -10119.682,E2 -10119.682} C_VEL
LIN {X 0,Y 418.234,Z 419.393,A -85,B 0,C 180,E1 -10122.322,E2 -10122.322} C_VEL
LIN {X 0,Y 418.24,Z 419.392,A -85,B 0,C 180,E1 -10125.109,E2 -10125.109} C_VEL
LIN {X 0,Y 418.269,Z 419.436,A -85,B 0,C 180,E1 -10127.591,E2 -10127.591} C_VEL
LIN {X 0,Y 420.072,Z 428.255,A -85,B 0,C 180,E1 -10130.524,E2 -10130.524} C_VEL
LIN {X 0,Y 421.446,Z 436.55,A -85,B 0,C 180,E1 -10133.106,E2 -10133.106} C_VEL
LIN {X 0,Y 420.598,Z 448.739,A -85,B 0,C 180,E1 -10136.536,E2 -10136.536} C_VEL
LIN {X 0,Y 419.935,Z 459.934,A -85,B 0,C 180,E1 -10139.585,E2 -10139.585} C_VEL
LIN {X 0,Y 419.218,Z 473.089,A -85,B 0,C 180,E1 -10143.087,E2 -10143.087} C_VEL
LIN {X 0,Y 418.694,Z 485.102,A -85,B 0,C 180,E1 -10146.243,E2 -10146.243} C_VEL
LIN {X 0,Y 418.129,Z 500.437,A -85,B 0,C 180,E1 -10150.265,E2 -10150.265} C_VEL
LIN {X 0,Y 417.785,Z 509.669,A -85,B 0,C 180,E1 -10152.681,E2 -10152.681} C_VEL
LIN {X 0,Y 419.405,Z 523.811,A -85,B 0,C 180,E1 -10153.129,E2 -10153.129} C_VEL
LIN {X 0,Y 420.309,Z 537.115,A -85,B 0,C 180,E1 -10153.735,E2 -10153.735} C_VEL
LIN {X 0,Y 420.839,Z 547.81,A -85,B 0,C 180,E1 -10154.378,E2 -10154.378} C_VEL
LIN {X 0,Y 420.014,Z 559.279,A -85,B 0,C 180,E1 -10155.216,E2 -10155.216} C_VEL
LIN {X 0,Y 419.29,Z 570.993,A -85,B 0,C 180,E1 -10156.305,E2 -10156.305} C_VEL
LIN {X 0,Y 418.79,Z 580.476,A -85,B 0,C 180,E1 -10157.399,E2 -10157.399} C_VEL
LIN {X 0,Y 418.178,Z 589.123,A -85,B 0,C 180,E1 -10158.611,E2 -10158.611} C_VEL
LIN {X 0,Y 417.735,Z 597.597,A -85,B 0,C 180,E1 -10160.07,E2 -10160.07} C_VEL
LIN {X 0,Y 417.537,Z 604.464,A -85,B 0,C 180,E1 -10161.531,E2 -10161.531} C_VEL
LIN {X 0,Y 417.475,Z 610.777,A -85,B 0,C 180,E1 -10163.232,E2 -10163.232} C_VEL
LIN {X 0,Y 417.569,Z 614.901,A -85,B 0,C 180,E1 -10164.689,E2 -10164.689} C_VEL
LIN {X 0,Y 417.673,Z 617.953,A -85,B 0,C 180,E1 -10166.141,E2 -10166.141} C_VEL
LIN {X 0,Y 417.652,Z 619.397,A -85,B 0,C 180,E1 -10167.106,E2 -10167.106} C_VEL
LIN {X 0,Y 417.671,Z 620.432,A -85,B 0,C 180,E1 -10168.072,E2 -10168.072} C_VEL
LIN {X 0,Y 417.884,Z 621.316,A -85,B 0,C 180,E1 -10170,E2 -10170} C_VEL
LIN {X 0,Y 417.671,Z 620.432,A -85,B 0,C 180,E1 -10171.929,E2 -10171.929} C_VEL
LIN {X 0,Y 417.652,Z 619.398,A -85,B 0,C 180,E1 -10172.894,E2 -10172.894} C_VEL
LIN {X 0,Y 417.673,Z 617.952,A -85,B 0,C 180,E1 -10173.859,E2 -10173.859} C_VEL
LIN {X 0,Y 417.568,Z 614.895,A -85,B 0,C 180,E1 -10175.312,E2 -10175.312} C_VEL
LIN {X 0,Y 417.477,Z 610.767,A -85,B 0,C 180,E1 -10176.768,E2 -10176.768} C_VEL
LIN {X 0,Y 417.538,Z 604.451,A -85,B 0,C 180,E1 -10178.469,E2 -10178.469} C_VEL
LIN {X 0,Y 417.736,Z 597.581,A -85,B 0,C 180,E1 -10179.93,E2 -10179.93} C_VEL
LIN {X 0,Y 418.178,Z 589.102,A -85,B 0,C 180,E1 -10181.389,E2 -10181.389} C_VEL
LIN {X 0,Y 418.793,Z 580.448,A -85,B 0,C 180,E1 -10182.601,E2 -10182.601} C_VEL
LIN {X 0,Y 419.292,Z 570.955,A -85,B 0,C 180,E1 -10183.695,E2 -10183.695} C_VEL
LIN {X 0,Y 420.011,Z 559.234,A -85,B 0,C 180,E1 -10184.784,E2 -10184.784} C_VEL
LIN {X 0,Y 420.847,Z 547.747,A -85,B 0,C 180,E1 -10185.622,E2 -10185.622} C_VEL
LIN {X 0,Y 420.208,Z 535.765,A -85,B 0,C 180,E1 -10186.331,E2 -10186.331} C_VEL
LIN {X 0,Y 419.221,Z 522.226,A -85,B 0,C 180,E1 -10186.927,E2 -10186.927} C_VEL
LIN {X 0,Y 417.807,Z 509.53,A -85,B 0,C 180,E1 -10187.318,E2 -10187.318} C_VEL
LIN {X 0,Y 418.158,Z 497.94,A -85,B 0,C 180,E1 -10190.385,E2 -10190.385} C_VEL
LIN {X 0,Y 418.695,Z 485.07,A -85,B 0,C 180,E1 -10193.757,E2 -10193.757} C_VEL
LIN {X 0,Y 419.194,Z 473.042,A -85,B 0,C 180,E1 -10196.915,E2 -10196.915} C_VEL
LIN {X 0,Y 419.914,Z 459.894,A -85,B 0,C 180,E1 -10200.417,E2 -10200.417} C_VEL
LIN {X 0,Y 420.57,Z 448.694,A -85,B 0,C 180,E1 -10203.467,E2 -10203.467} C_VEL
LIN {X 0,Y 421.44,Z 436.742,A -85,B 0,C 180,E1 -10206.826,E2 -10206.826} C_VEL
LIN {X 0,Y 420.271,Z 429.243,A -85,B 0,C 180,E1 -10209.144,E2 -10209.144} C_VEL
LIN {X 0,Y 418.372,Z 419.945,A -85,B 0,C 180,E1 -10212.217,E2 -10212.217} C_VEL
LIN {X 0,Y 418.27,Z 419.385,A -85,B 0,C 180,E1 -10212.449,E2 -10212.449} C_VEL
LIN {X 0,Y 418.242,Z 419.388,A -85,B 0,C 180,E1 -10215.109,E2 -10215.109} C_VEL
LIN {X 0,Y 418.245,Z 419.388,A -85,B 0,C 180,E1 -10217.767,E2 -10217.767} C_VEL
LIN {X 0,Y 418.26,Z 419.385,A -85,B 0,C 180,E1 -10220.619,E2 -10220.619} C_VEL
LIN {X 0,Y 418.249,Z 419.389,A -85,B 0,C 180,E1 -10223.976,E2 -10223.976} C_VEL
LIN {X 0,Y 418.261,Z 419.383,A -85,B 0,C 180,E1 -10227.156,E2 -10227.156} C_VEL
LIN {X 0,Y 418.272,Z 419.381,A -85,B 0,C 180,E1 -10230.896,E2 -10230.896} C_VEL
LIN {X 0,Y 418.271,Z 419.386,A -85,B 0,C 180,E1 -10234.096,E2 -10234.096} C_VEL
LIN {X 0,Y 418.235,Z 419.387,A -85,B 0,C 180,E1 -10237.264,E2 -10237.264} C_VEL
LIN {X 0,Y 418.287,Z 419.382,A -85,B 0,C 180,E1 -10240.364,E2 -10240.364} C_VEL
LIN {X 0,Y 418.321,Z 419.378,A -85,B 0,C 180,E1 -10243.405,E2 -10243.405} C_VEL
LIN {X 0,Y 418.359,Z 419.37,A -85,B 0,C 180,E1 -10246.994,E2 -10246.994} C_VEL
LIN {X 0,Y 418.345,Z 419.374,A -85,B 0,C 180,E1 -10250.329,E2 -10250.329} C_VEL
LIN {X 0,Y 418.483,Z 419.358,A -85,B 0,C 180,E1 -10253.249,E2 -10253.249} C_VEL
LIN {X 0,Y 418.345,Z 419.374,A -85,B 0,C 180,E1 -10255.182,E2 -10255.182} C_VEL
LIN {X 0,Y 418.55,Z 419.349,A -85,B 0,C 180,E1 -10258.076,E2 -10258.076} C_VEL
LIN {X 0,Y 418.677,Z 419.333,A -85,B 0,C 180,E1 -10260,E2 -10260} C_VEL
LIN {X 0,Y 418.506,Z 419.353,A -85,B 0,C 180,E1 -10262.888,E2 -10262.888} C_VEL
LIN {X 0,Y 418.479,Z 419.356,A -85,B 0,C 180,E1 -10266.643,E2 -10266.643} C_VEL
LIN {X 0,Y 418.346,Z 419.376,A -85,B 0,C 180,E1 -10269.671,E2 -10269.671} C_VEL
LIN {X 0,Y 418.359,Z 419.373,A -85,B 0,C 180,E1 -10273.006,E2 -10273.006} C_VEL
LIN {X 0,Y 418.317,Z 419.376,A -85,B 0,C 180,E1 -10276.736,E2 -10276.736} C_VEL
LIN {X 0,Y 418.275,Z 419.384,A -85,B 0,C 180,E1 -10279.79,E2 -10279.79} C_VEL
LIN {X 0,Y 418.242,Z 419.387,A -85,B 0,C 180,E1 -10282.736,E2 -10282.736} C_VEL
LIN {X 0,Y 418.275,Z 419.382,A -85,B 0,C 180,E1 -10285.904,E2 -10285.904} C_VEL
LIN {X 0,Y 418.268,Z 419.386,A -85,B 0,C 180,E1 -10289.162,E2 -10289.162} C_VEL
LIN {X 0,Y 418.261,Z 419.385,A -85,B 0,C 180,E1 -10292.844,E2 -10292.844} C_VEL
LIN {X 0,Y 418.248,Z 419.385,A -85,B 0,C 180,E1 -10296.238,E2 -10296.238} C_VEL
LIN {X 0,Y 418.25,Z 419.386,A -85,B 0,C 180,E1 -10299.682,E2 -10299.682} C_VEL
LIN {X 0,Y 418.235,Z 419.386,A -85,B 0,C 180,E1 -10302.322,E2 -10302.322} C_VEL
LIN {X 0,Y 418.265,Z 419.387,A -85,B 0,C 180,E1 -10305.112,E2 -10305.112} C_VEL
LIN {X 0,Y 418.296,Z 419.379,A -85,B 0,C 180,E1 -10307.773,E2 -10307.773} C_VEL
LIN {X 0,Y 418.27,Z 419.383,A -85,B 0,C 180,E1 -10311.56,E2 -10311.56} C_VEL
LIN {X 0,Y 418.262,Z 419.386,A -85,B 0,C 180,E1 -10315.159,E2 -10315.159} C_VEL
LIN {X 0,Y 418.249,Z 419.385,A -85,B 0,C 180,E1 -10317.472,E2 -10317.472} C_VEL
LIN {X 0,Y 418.272,Z 419.386,A -85,B 0,C 180,E1 -10320.895,E2 -10320.895} C_VEL
LIN {X 0,Y 418.275,Z 419.382,A -85,B 0,C 180,E1 -10324.096,E2 -10324.096} C_VEL
LIN {X 0,Y 418.242,Z 419.387,A -85,B 0,C 180,E1 -10327.264,E2 -10327.264} C_VEL
LIN {X 0,Y 418.287,Z 419.383,A -85,B 0,C 180,E1 -10330.364,E2 -10330.364} C_VEL
LIN {X 0,Y 418.359,Z 419.433,A -85,B 0,C 180,E1 -10333.579,E2 -10333.579} C_VEL
LIN {X 0,Y 421.812,Z 430.999,A -85,B 0,C 180,E1 -10334.415,E2 -10334.415} C_VEL
LIN {X 0,Y 422.746,Z 435.064,A -85,B 0,C 180,E1 -10334.748,E2 -10334.748} C_VEL
LIN {X 0,Y 422.129,Z 446.358,A -85,B 0,C 180,E1 -10335.661,E2 -10335.661} C_VEL
LIN {X 0,Y 421.466,Z 456.913,A -85,B 0,C 180,E1 -10336.745,E2 -10336.745} C_VEL
LIN {X 0,Y 420.861,Z 466.384,A -85,B 0,C 180,E1 -10337.951,E2 -10337.951} C_VEL
LIN {X 0,Y 420.265,Z 474.137,A -85,B 0,C 180,E1 -10339.156,E2 -10339.156} C_VEL
LIN {X 0,Y 419.612,Z 481.714,A -85,B 0,C 180,E1 -10340.601,E2 -10340.601} C_VEL
LIN {X 0,Y 419.257,Z 486.987,A -85,B 0,C 180,E1 -10341.842,E2 -10341.842} C_VEL
LIN {X 0,Y 418.956,Z 491.836,A -85,B 0,C 180,E1 -10343.256,E2 -10343.256} C_VEL
LIN {X 0,Y 418.529,Z 495.726,A -85,B 0,C 180,E1 -10344.701,E2 -10344.701} C_VEL
LIN {X 0,Y 418.254,Z 498.592,A -85,B 0,C 180,E1 -10346.146,E2 -10346.146} C_VEL
LIN {X 0,Y 418.102,Z 499.969,A -85,B 0,C 180,E1 -10347.109,E2 -10347.109} C_VEL
LIN {X 0,Y 418.121,Z 500.928,A -85,B 0,C 180,E1 -10348.073,E2 -10348.073} C_VEL
LIN {X 0,Y 418.121,Z 501.749,A -85,B 0,C 180,E1 -10350,E2 -10350} C_VEL
LIN {X 0,Y 418.052,Z 501.577,A -85,B 0,C 180,E1 -10350.963,E2 -10350.963} C_VEL
LIN {X 0,Y 418.12,Z 501.003,A -85,B 0,C 180,E1 -10351.926,E2 -10351.926} C_VEL
LIN {X 0,Y 418.246,Z 498.743,A -85,B 0,C 180,E1 -10353.854,E2 -10353.854} C_VEL
LIN {X 0,Y 418.523,Z 495.934,A -85,B 0,C 180,E1 -10355.299,E2 -10355.299} C_VEL
LIN {X 0,Y 418.933,Z 492.116,A -85,B 0,C 180,E1 -10356.744,E2 -10356.744} C_VEL
LIN {X 0,Y 419.035,Z 489.689,A -85,B 0,C 180,E1 -10357.499,E2 -10357.499} C_VEL
LIN {X 0,Y 418.504,Z 487.229,A -85,B 0,C 180,E1 -10358.233,E2 -10358.233} C_VEL
LIN {X 0,Y 416.04,Z 482.99,A -85,B 0,C 180,E1 -10359.42,E2 -10359.42} C_VEL
LIN {X 0,Y 413.743,Z 478.079,A -85,B 0,C 180,E1 -10360.563,E2 -10360.563} C_VEL
LIN {X 0,Y 413.463,Z 474.571,A -85,B 0,C 180,E1 -10361.218,E2 -10361.218} C_VEL
LIN {X 0,Y 414.059,Z 466.328,A -85,B 0,C 180,E1 -10362.498,E2 -10362.498} C_VEL
LIN {X 0,Y 414.745,Z 456.635,A -85,B 0,C 180,E1 -10363.723,E2 -10363.723} C_VEL
LIN {X 0,Y 415.338,Z 447.078,A -85,B 0,C 180,E1 -10364.703,E2 -10364.703} C_VEL
LIN {X 0,Y 415.927,Z 436.103,A -85,B 0,C 180,E1 -10365.604,E2 -10365.604} C_VEL
LIN {X 0,Y 412.878,Z 425.4,A -85,B 0,C 180,E1 -10366.464,E2 -10366.464} C_VEL
LIN {X 0,Y 411.27,Z 420.256,A -85,B 0,C 180,E1 -10366.835,E2 -10366.835} C_VEL
LIN {X 0,Y 411.233,Z 420.263,A -85,B 0,C 180,E1 -10369.987,E2 -10369.987} C_VEL
LIN {X 0,Y 411.206,Z 420.266,A -85,B 0,C 180,E1 -10373.147,E2 -10373.147} C_VEL
LIN {X 0,Y 411.241,Z 420.257,A -85,B 0,C 180,E1 -10376.381,E2 -10376.381} C_VEL
LIN {X 0,Y 411.203,Z 420.263,A -85,B 0,C 180,E1 -10379.713,E2 -10379.713} C_VEL
LIN {X 0,Y 411.209,Z 420.266,A -85,B 0,C 180,E1 -10383.156,E2 -10383.156} C_VEL
LIN {X 0,Y 411.199,Z 420.264,A -85,B 0,C 180,E1 -10386.553,E2 -10386.553} C_VEL
LIN {X 0,Y 411.232,Z 420.259,A -85,B 0,C 180,E1 -10389.73,E2 -10389.73} C_VEL
LIN {X 0,Y 411.231,Z 420.264,A -85,B 0,C 180,E1 -10393.126,E2 -10393.126} C_VEL
LIN {X 0,Y 411.179,Z 420.264,A -85,B 0,C 180,E1 -10395.88,E2 -10395.88} C_VEL
LIN {X 0,Y 411.167,Z 420.271,A -85,B 0,C 180,E1 -10398.771,E2 -10398.771} C_VEL
LIN {X 0,Y 411.208,Z 420.261,A -85,B 0,C 180,E1 -10401.831,E2 -10401.831} C_VEL
LIN {X 0,Y 411.213,Z 420.264,A -85,B 0,C 180,E1 -10405.121,E2 -10405.121} C_VEL
LIN {X 0,Y 411.168,Z 420.266,A -85,B 0,C 180,E1 -10408.003,E2 -10408.003} C_VEL
LIN {X 0,Y 411.22,Z 420.26,A -85,B 0,C 180,E1 -10411.41,E2 -10411.41} C_VEL
LIN {X 0,Y 411.239,Z 420.257,A -85,B 0,C 180,E1 -10413.619,E2 -10413.619} C_VEL
LIN {X 0,Y 411.204,Z 420.266,A -85,B 0,C 180,E1 -10416.852,E2 -10416.852} C_VEL
LIN {X 0,Y 411.218,Z 420.261,A -85,B 0,C 180,E1 -10420.05,E2 -10420.05} C_VEL
LIN {X 0,Y 411.265,Z 420.256,A -85,B 0,C 180,E1 -10423.131,E2 -10423.131} C_VEL
LIN {X 0,Y 411.316,Z 420.251,A -85,B 0,C 180,E1 -10426.891,E2 -10426.891} C_VEL
LIN {X 0,Y 411.298,Z 420.253,A -85,B 0,C 180,E1 -10430.161,E2 -10430.161} C_VEL
LIN {X 0,Y 411.445,Z 420.233,A -85,B 0,C 180,E1 -10433.133,E2 -10433.133} C_VEL
LIN {X 0,Y 411.313,Z 420.249,A -85,B 0,C 180,E1 -10435.099,E2 -10435.099} C_VEL
LIN {X 0,Y 411.517,Z 420.225,A -85,B 0,C 180,E1 -10438.043,E2 -10438.043} C_VEL
LIN {X 0,Y 411.645,Z 420.209,A -85,B 0,C 180,E1 -10440,E2 -10440} C_VEL
LIN {X 0,Y 411.47,Z 420.23,A -85,B 0,C 180,E1 -10442.937,E2 -10442.937} C_VEL
LIN {X 0,Y 411.474,Z 420.23,A -85,B 0,C 180,E1 -10445.882,E2 -10445.882} C_VEL
LIN {X 0,Y 411.322,Z 420.249,A -85,B 0,C 180,E1 -10448.846,E2 -10448.846} C_VEL
LIN {X 0,Y 411.301,Z 420.252,A -85,B 0,C 180,E1 -10451.832,E2 -10451.832} C_VEL
LIN {X 0,Y 411.265,Z 420.255,A -85,B 0,C 180,E1 -10454.852,E2 -10454.852} C_VEL
LIN {X 0,Y 411.256,Z 420.259,A -85,B 0,C 180,E1 -10457.915,E2 -10457.915} C_VEL
LIN {X 0,Y 411.199,Z 420.263,A -85,B 0,C 180,E1 -10461.034,E2 -10461.034} C_VEL
LIN {X 0,Y 411.222,Z 420.264,A -85,B 0,C 180,E1 -10464.216,E2 -10464.216} C_VEL
LIN {X 0,Y 411.261,Z 420.256,A -85,B 0,C 180,E1 -10467.478,E2 -10467.478} C_VEL
LIN {X 0,Y 411.191,Z 420.263,A -85,B 0,C 180,E1 -10470.848,E2 -10470.848} C_VEL
LIN {X 0,Y 411.208,Z 420.264,A -85,B 0,C 180,E1 -10474.333,E2 -10474.333} C_VEL
LIN {X 0,Y 411.202,Z 420.267,A -85,B 0,C 180,E1 -10477.973,E2 -10477.973} C_VEL
LIN {X 0,Y 411.166,Z 420.267,A -85,B 0,C 180,E1 -10481.229,E2 -10481.229} C_VEL
LIN {X 0,Y 411.181,Z 420.271,A -85,B 0,C 180,E1 -10484.49,E2 -10484.49} C_VEL
LIN {X 0,Y 411.254,Z 420.452,A -85,B 0,C 180,E1 -10487.293,E2 -10487.293} C_VEL
LIN {X 0,Y 413.202,Z 429.966,A -85,B 0,C 180,E1 -10490.518,E2 -10490.518} C_VEL
LIN {X 0,Y 414.449,Z 437.293,A -85,B 0,C 180,E1 -10492.845,E2 -10492.845} C_VEL
LIN {X 0,Y 414.043,Z 443.847,A -85,B 0,C 180,E1 -10494.752,E2 -10494.752} C_VEL
LIN {X 0,Y 413.243,Z 456.262,A -85,B 0,C 180,E1 -10498.25,E2 -10498.25} C_VEL
LIN {X 0,Y 412.367,Z 470.032,A -85,B 0,C 180,E1 -10502.014,E2 -10502.014} C_VEL
LIN {X 0,Y 411.752,Z 482.166,A -85,B 0,C 180,E1 -10505.28,E2 -10505.28} C_VEL
LIN {X 0,Y 411.238,Z 493.972,A -85,B 0,C 180,E1 -10508.443,E2 -10508.443} C_VEL
LIN {X 0,Y 410.856,Z 505.516,A -85,B 0,C 180,E1 -10511.551,E2 -10511.551} C_VEL
LIN {X 0,Y 410.743,Z 508.498,A -85,B 0,C 180,E1 -10512.363,E2 -10512.363} C_VEL
LIN {X 0,Y 412.39,Z 523.303,A -85,B 0,C 180,E1 -10512.851,E2 -10512.851} C_VEL
LIN {X 0,Y 413.306,Z 536.077,A -85,B 0,C 180,E1 -10513.452,E2 -10513.452} C_VEL
LIN {X 0,Y 413.841,Z 548.575,A -85,B 0,C 180,E1 -10514.233,E2 -10514.233} C_VEL
LIN {X 0,Y 412.902,Z 561.145,A -85,B 0,C 180,E1 -10515.208,E2 -10515.208} C_VEL
LIN {X 0,Y 412.148,Z 572.254,A -85,B 0,C 180,E1 -10516.319,E2 -10516.319} C_VEL
LIN {X 0,Y 411.651,Z 581.285,A -85,B 0,C 180,E1 -10517.427,E2 -10517.427} C_VEL
LIN {X 0,Y 411.06,Z 589.622,A -85,B 0,C 180,E1 -10518.661,E2 -10518.661} C_VEL
LIN {X 0,Y 410.647,Z 597.844,A -85,B 0,C 180,E1 -10520.146,E2 -10520.146} C_VEL
LIN {X 0,Y 410.458,Z 604.474,A -85,B 0,C 180,E1 -10521.632,E2 -10521.632} C_VEL
LIN {X 0,Y 410.423,Z 610.333,A -85,B 0,C 180,E1 -10523.306,E2 -10523.306} C_VEL
LIN {X 0,Y 410.581,Z 615.007,A -85,B 0,C 180,E1 -10525.09,E2 -10525.09} C_VEL
LIN {X 0,Y 410.636,Z 616.944,A -85,B 0,C 180,E1 -10526.075,E2 -10526.075} C_VEL
LIN {X 0,Y 410.609,Z 618.389,A -85,B 0,C 180,E1 -10527.057,E2 -10527.057} C_VEL
LIN {X 0,Y 410.633,Z 619.426,A -85,B 0,C 180,E1 -10528.038,E2 -10528.038} C_VEL
LIN {X 0,Y 410.861,Z 620.312,A -85,B 0,C 180,E1 -10530,E2 -10530} C_VEL
LIN {X 0,Y 410.633,Z 619.425,A -85,B 0,C 180,E1 -10531.962,E2 -10531.962} C_VEL
LIN {X 0,Y 410.61,Z 618.389,A -85,B 0,C 180,E1 -10532.943,E2 -10532.943} C_VEL
LIN {X 0,Y 410.636,Z 616.943,A -85,B 0,C 180,E1 -10533.926,E2 -10533.926} C_VEL
LIN {X 0,Y 410.488,Z 613.878,A -85,B 0,C 180,E1 -10535.403,E2 -10535.403} C_VEL
LIN {X 0,Y 410.423,Z 609.75,A -85,B 0,C 180,E1 -10536.885,E2 -10536.885} C_VEL
LIN {X 0,Y 410.476,Z 603.428,A -85,B 0,C 180,E1 -10538.616,E2 -10538.616} C_VEL
LIN {X 0,Y 410.689,Z 596.556,A -85,B 0,C 180,E1 -10540.102,E2 -10540.102} C_VEL
LIN {X 0,Y 411.155,Z 588.075,A -85,B 0,C 180,E1 -10541.587,E2 -10541.587} C_VEL
LIN {X 0,Y 411.874,Z 578.209,A -85,B 0,C 180,E1 -10542.969,E2 -10542.969} C_VEL
LIN {X 0,Y 412.318,Z 569.925,A -85,B 0,C 180,E1 -10543.932,E2 -10543.932} C_VEL
LIN {X 0,Y 413.126,Z 558.211,A -85,B 0,C 180,E1 -10545.036,E2 -10545.036} C_VEL
LIN {X 0,Y 413.911,Z 546.712,A -85,B 0,C 180,E1 -10545.89,E2 -10545.89} C_VEL
LIN {X 0,Y 413.211,Z 534.715,A -85,B 0,C 180,E1 -10546.616,E2 -10546.616} C_VEL
LIN {X 0,Y 412.216,Z 521.593,A -85,B 0,C 180,E1 -10547.208,E2 -10547.208} C_VEL
LIN {X 0,Y 410.782,Z 508.403,A -85,B 0,C 180,E1 -10547.653,E2 -10547.653} C_VEL
LIN {X 0,Y 411.136,Z 495.892,A -85,B 0,C 180,E1 -10551.038,E2 -10551.038} C_VEL
LIN {X 0,Y 411.67,Z 484.121,A -85,B 0,C 180,E1 -10554.188,E2 -10554.188} C_VEL
LIN {X 0,Y 412.271,Z 471.532,A -85,B 0,C 180,E1 -10557.57,E2 -10557.57} C_VEL
LIN {X 0,Y 413.104,Z 458.15,A -85,B 0,C 180,E1 -10561.219,E2 -10561.219} C_VEL
LIN {X 0,Y 413.86,Z 445.832,A -85,B 0,C 180,E1 -10564.673,E2 -10564.673} C_VEL
LIN {X 0,Y 414.465,Z 438.513,A -85,B 0,C 180,E1 -10566.777,E2 -10566.777} C_VEL
LIN {X 0,Y 413.939,Z 434.166,A -85,B 0,C 180,E1 -10568.122,E2 -10568.122} C_VEL
LIN {X 0,Y 412.349,Z 425.83,A -85,B 0,C 180,E1 -10570.843,E2 -10570.843} C_VEL
LIN {X 0,Y 411.205,Z 420.267,A -85,B 0,C 180,E1 -10572.78,E2 -10572.78} C_VEL
LIN {X 0,Y 411.175,Z 420.269,A -85,B 0,C 180,E1 -10575.88,E2 -10575.88} C_VEL
LIN {X 0,Y 411.168,Z 420.273,A -85,B 0,C 180,E1 -10578.772,E2 -10578.772} C_VEL
LIN {X 0,Y 411.203,Z 420.267,A -85,B 0,C 180,E1 -10582.027,E2 -10582.027} C_VEL
LIN {X 0,Y 411.209,Z 420.264,A -85,B 0,C 180,E1 -10585.667,E2 -10585.667} C_VEL
LIN {X 0,Y 411.192,Z 420.263,A -85,B 0,C 180,E1 -10589.153,E2 -10589.153} C_VEL
LIN {X 0,Y 411.262,Z 420.256,A -85,B 0,C 180,E1 -10592.522,E2 -10592.522} C_VEL
LIN {X 0,Y 411.223,Z 420.264,A -85,B 0,C 180,E1 -10595.784,E2 -10595.784} C_VEL
LIN {X 0,Y 411.2,Z 420.262,A -85,B 0,C 180,E1 -10598.966,E2 -10598.966} C_VEL
LIN {X 0,Y 411.257,Z 420.259,A -85,B 0,C 180,E1 -10602.085,E2 -10602.085} C_VEL
LIN {X 0,Y 411.266,Z 420.254,A -85,B 0,C 180,E1 -10605.148,E2 -10605.148} C_VEL
LIN {X 0,Y 411.302,Z 420.252,A -85,B 0,C 180,E1 -10608.168,E2 -10608.168} C_VEL
LIN {X 0,Y 411.441,Z 420.234,A -85,B 0,C 180,E1 -10612.191,E2 -10612.191} C_VEL
LIN {X 0,Y 411.475,Z 420.231,A -85,B 0,C 180,E1 -10614.118,E2 -10614.118} C_VEL
LIN {X 0,Y 411.519,Z 420.225,A -85,B 0,C 180,E1 -10618.043,E2 -10618.043} C_VEL
LIN {X 0,Y 411.646,Z 420.209,A -85,B 0,C 180,E1 -10620,E2 -10620} C_VEL
LIN {X 0,Y 411.462,Z 420.23,A -85,B 0,C 180,E1 -10622.937,E2 -10622.937} C_VEL
LIN {X 0,Y 411.441,Z 420.232,A -85,B 0,C 180,E1 -10626.643,E2 -10626.643} C_VEL
LIN {X 0,Y 411.324,Z 420.248,A -85,B 0,C 180,E1 -10628.846,E2 -10628.846} C_VEL
LIN {X 0,Y 411.303,Z 420.252,A -85,B 0,C 180,E1 -10631.832,E2 -10631.832} C_VEL
LIN {X 0,Y 411.267,Z 420.255,A -85,B 0,C 180,E1 -10634.853,E2 -10634.853} C_VEL
LIN {X 0,Y 411.257,Z 420.257,A -85,B 0,C 180,E1 -10637.915,E2 -10637.915} C_VEL
LIN {X 0,Y 411.2,Z 420.265,A -85,B 0,C 180,E1 -10641.034,E2 -10641.034} C_VEL
LIN {X 0,Y 411.23,Z 420.259,A -85,B 0,C 180,E1 -10644.215,E2 -10644.215} C_VEL
LIN {X 0,Y 411.262,Z 420.259,A -85,B 0,C 180,E1 -10647.478,E2 -10647.478} C_VEL
LIN {X 0,Y 411.193,Z 420.265,A -85,B 0,C 180,E1 -10650.848,E2 -10650.848} C_VEL
LIN {X 0,Y 411.209,Z 420.261,A -85,B 0,C 180,E1 -10654.333,E2 -10654.333} C_VEL
LIN {X 0,Y 411.196,Z 420.263,A -85,B 0,C 180,E1 -10657.974,E2 -10657.974} C_VEL
LIN {X 0,Y 411.168,Z 420.271,A -85,B 0,C 180,E1 -10661.228,E2 -10661.228} C_VEL
LIN {X 0,Y 411.192,Z 420.264,A -85,B 0,C 180,E1 -10664.489,E2 -10664.489} C_VEL
LIN {X 0,Y 411.232,Z 420.262,A -85,B 0,C 180,E1 -10667.297,E2 -10667.297} C_VEL
LIN {X 0,Y 411.235,Z 420.262,A -85,B 0,C 180,E1 -10670.778,E2 -10670.778} C_VEL
LIN {X 0,Y 411.202,Z 420.264,A -85,B 0,C 180,E1 -10674.471,E2 -10674.471} C_VEL
LIN {X 0,Y 411.21,Z 420.266,A -85,B 0,C 180,E1 -10676.873,E2 -10676.873} C_VEL
LIN {X 0,Y 411.236,Z 420.262,A -85,B 0,C 180,E1 -10680.644,E2 -10680.644} C_VEL
LIN {X 0,Y 411.241,Z 420.257,A -85,B 0,C 180,E1 -10683.619,E2 -10683.619} C_VEL
LIN {X 0,Y 411.207,Z 420.266,A -85,B 0,C 180,E1 -10686.852,E2 -10686.852} C_VEL
LIN {X 0,Y 411.218,Z 420.261,A -85,B 0,C 180,E1 -10690.05,E2 -10690.05} C_VEL
LIN {X 0,Y 411.272,Z 420.257,A -85,B 0,C 180,E1 -10693.27,E2 -10693.27} C_VEL
LIN {X 0,Y 414.862,Z 432.038,A -85,B 0,C 180,E1 -10694.147,E2 -10694.147} C_VEL
LIN {X 0,Y 415.83,Z 435.496,A -85,B 0,C 180,E1 -10694.444,E2 -10694.444} C_VEL
LIN {X 0,Y 415.534,Z 444.611,A -85,B 0,C 180,E1 -10695.178,E2 -10695.178} C_VEL
LIN {X 0,Y 414.853,Z 454.661,A -85,B 0,C 180,E1 -10696.155,E2 -10696.155} C_VEL
LIN {X 0,Y 414.257,Z 463.858,A -85,B 0,C 180,E1 -10697.259,E2 -10697.259} C_VEL
LIN {X 0,Y 413.635,Z 472.232,A -85,B 0,C 180,E1 -10698.484,E2 -10698.484} C_VEL
LIN {X 0,Y 412.89,Z 480.362,A -85,B 0,C 180,E1 -10699.952,E2 -10699.952} C_VEL
LIN {X 0,Y 412.347,Z 486.489,A -85,B 0,C 180,E1 -10701.321,E2 -10701.321} C_VEL
LIN {X 0,Y 411.981,Z 492.842,A -85,B 0,C 180,E1 -10703.142,E2 -10703.142} C_VEL
LIN {X 0,Y 411.534,Z 496.732,A -85,B 0,C 180,E1 -10704.61,E2 -10704.61} C_VEL
LIN {X 0,Y 411.242,Z 499.598,A -85,B 0,C 180,E1 -10706.08,E2 -10706.08} C_VEL
LIN {X 0,Y 411.083,Z 500.975,A -85,B 0,C 180,E1 -10707.06,E2 -10707.06} C_VEL
LIN {X 0,Y 411.1,Z 501.934,A -85,B 0,C 180,E1 -10708.041,E2 -10708.041} C_VEL
LIN {X 0,Y 411.108,Z 502.752,A -85,B 0,C 180,E1 -10710,E2 -10710} C_VEL
LIN {X 0,Y 411.099,Z 502.008,A -85,B 0,C 180,E1 -10711.959,E2 -10711.959} C_VEL
